KUKA KRL program: Enlargedx2Test.src

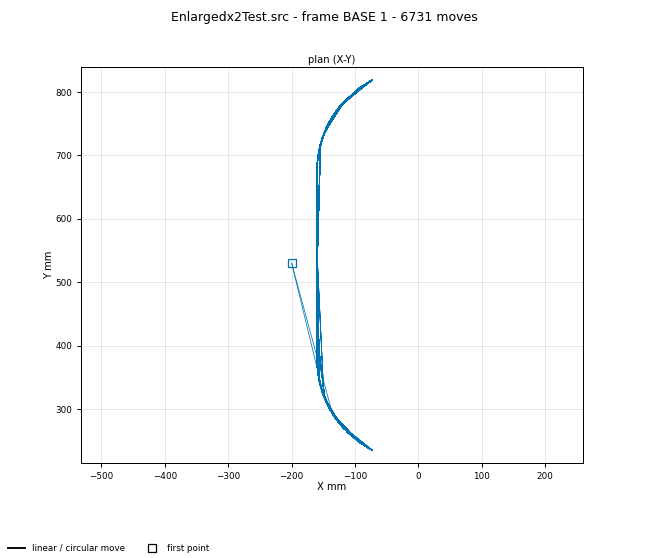
[picture p0: tool path of Enlargedx2Test.src in frame BASE 1, 6731 of 6732 moves have a stored position in this frame; points joined in program order, loops and branches not executed]
&ACCESS RVEO
&REL 11
&PARAM TEMPLATE = C:\KRC\Roboter\Template\vorgabe
&PARAM EDITMASK = *
DEF variable_helical2( )
;FOLD INI
  ;FOLD BASISTECH INI
    GLOBAL INTERRUPT DECL 3 WHEN $STOPMESS==TRUE DO IR_STOPM ( )
    INTERRUPT ON 3
    BAS (#INITMOV,0 )
  ;ENDFOLD (BASISTECH INI)
 ;FOLD USER INI


    ;Make your modifications here
  ;ENDFOLD (USER INI)
;ENDFOLD (INI)
ACTION(#AXIS_RESET,34,1000,#NOERROR,ERROR_CODE)
;FOLD PTP HOME  Vel= 100 % DEFAULT;%{PE}%MKUKATPBASIS,%CMOVE,%VPTP,%P 1:PTP, 2:HOME, 3:, 5:100, 7:DEFAULT
$BWDSTART = FALSE
PDAT_ACT=PDEFAULT
FDAT_ACT=FHOME
BAS (#PTP_PARAMS,100 )
$H_POS=XHOME
PTP  XHOME
;ENDFOLD
BAS(#TOOL,1)
BAS(#BASE,1)
$VEL_AXIS[1]=100
$VEL_AXIS[2]=100
$VEL_AXIS[3]=100
$VEL_AXIS[4]=100
$VEL_AXIS[5]=100
$VEL_AXIS[6]=100
$VEL_EXTAX[1]=100
$VEL_EXTAX[2]=100

$ACC_AXIS[1]=100
$ACC_AXIS[2]=100
$ACC_AXIS[3]=100
$ACC_AXIS[4]=100
$ACC_AXIS[5]=100
$ACC_AXIS[6]=100
$ACC_EXTAX[1]=100
$ACC_EXTAX[2]=100

;;;;;;;;; postprocessing parameters (date 2024-01-29T17:09:42.519984)
; qxconst: -159.99
; qxconstarcys: -152.5,146.5
; qE3offset: 0.00
; qyoffset: 530.00
; qswitchsplit: 3
; qthinningtol: 0.2010
;;;;;;;;;

SLIN {X  -200.000, Y  +530.000, Z    +0.000, A    +0.000, E1    +0.000, E3    +0.000, E4    +0.000}

SLIN {X  -135.697, Y  +292.747, Z    +0.000, E1   +74.259, E3  -294.688}
HALT
SPLINE
SPL {X  -132.590, Y  +287.964, Z    +0.000, E1   +73.910, E3  -289.659}
SPL {X  -129.541, Y  +283.606, Z    +0.000, E1   +73.551, E3  -285.019}
SPL {X  -126.457, Y  +279.493, Z    +0.000, E1   +73.175, E3  -280.620}
SPL {X  -122.770, Y  +274.912, Z    +0.000, E1   +72.712, E3  -275.765}
SPL {X  -119.156, Y  +270.736, Z    +0.000, E1   +72.213, E3  -271.415}
SPL {X  -117.531, Y  +268.949, Z    +0.000, E1   +71.964, E3  -269.600}
SPL {X   -74.907, Y  +236.129, Z    +0.000, E1   +61.720, E3  -192.564}
SPL {X   -72.759, Y  +235.012, Z    +0.000, E1   +56.036, E3   -20.886}
ENDSPLINE

SPLINE
SPL {X  -110.316, Y  +261.624, Z    +0.000, E1   +58.739, E3   +51.186}
SPL {X  -136.558, Y  +294.141, Z    +0.000, E1   +54.887, E3   +72.984}
SPL {X  -153.807, Y  +333.452, Z    +0.000, E1   +40.945, E3   +83.380}
SPL {X  -158.168, Y  +353.421, Z    +0.000, E1   +27.296, E3   +85.774}
SPL {X  -159.556, Y  +365.719, Z    +0.000, E1   +15.845, E3   +86.575}
SPL {X  -159.982, Y  +375.924, Z    +0.000, E1    +4.476, E3   +86.877}
SPL {X  -159.990, Y  +379.800, Z    +0.000, E1    -0.377, E3   +86.905}
SPL {X  -159.990, Y  +383.422, Z    +0.000, E1   -10.730, E3   +86.948}
SPL {X  -159.990, Y  +387.978, Z    +0.000, E1   -23.882, E3   +87.101}
SPL {X  -159.990, Y  +394.494, Z    +0.000, E1   -40.961, E3   +87.482}
SPL {X  -159.990, Y  +400.492, Z    +0.000, E1   -51.837, E3   +88.006}
SPL {X  -159.990, Y  +409.662, Z    +0.000, E1   -61.705, E3   +89.117}
SPL {X  -159.990, Y  +434.697, Z    +0.000, E1   -71.504, E3   +94.137}
SPL {X  -159.990, Y  +521.523, Z    +0.000, E1   -76.035, E3  +120.417}
SPL {X  -154.459, Y  +718.205, Z    +0.000, E1   -76.329, E3  +202.213}
SPL {X  -151.356, Y  +728.349, Z    +0.000, E1   -76.056, E3  +210.428}
SPL {X  -147.124, Y  +739.360, Z    +0.000, E1   -75.690, E3  +220.024}
SPL {X  -142.861, Y  +748.524, Z    +0.000, E1   -75.261, E3  +228.709}
SPL {X  -138.117, Y  +757.250, Z    +0.000, E1   -74.803, E3  +237.313}
SPL {X  -133.491, Y  +764.686, Z    +0.000, E1   -74.276, E3  +245.054}
SPL {X  -130.530, Y  +769.013, Z    +0.000, E1   -73.929, E3  +249.636}
SPL {X  -127.734, Y  +772.837, Z    +0.000, E1   -73.601, E3  +253.688}
SPL {X  -124.765, Y  +776.652, Z    +0.000, E1   -73.233, E3  +257.722}
SPL {X  -121.376, Y  +780.734, Z    +0.000, E1   -72.804, E3  +261.984}
SPL {X  -118.281, Y  +784.233, Z    +0.000, E1   -72.371, E3  +265.552}
SPL {X   -72.391, Y  +819.176, Z    +0.000, E1   -59.867, E3  +361.438}
ENDSPLINE

SPLINE
SPL {X   -92.809, Y  +806.820, Z    +0.000, E1   -56.994, E3  +554.233}
SPL {X  -120.521, Y  +781.721, Z    +0.000, E1   -56.766, E3  +590.332}
SPL {X  -143.482, Y  +747.279, Z    +0.000, E1   -50.227, E3  +608.345}
SPL {X  -154.118, Y  +719.449, Z    +0.000, E1   -38.836, E3  +614.924}
SPL {X  -158.958, Y  +694.646, Z    +0.000, E1   -21.132, E3  +617.775}
SPL {X  -159.960, Y  +679.609, Z    +0.000, E1    -6.021, E3  +618.475}
SPL {X  -159.990, Y  +674.508, Z    +0.000, E1    -0.018, E3  +618.534}
SPL {X  -159.990, Y  +672.787, Z    +0.000, E1    +4.022, E3  +618.546}
SPL {X  -159.990, Y  +669.267, Z    +0.000, E1   +13.665, E3  +618.616}
SPL {X  -159.990, Y  +665.069, Z    +0.000, E1   +25.376, E3  +618.788}
SPL {X  -159.990, Y  +657.821, Z    +0.000, E1   +42.408, E3  +619.290}
SPL {X  -159.990, Y  +645.368, Z    +0.000, E1   +59.257, E3  +620.747}
SPL {X  -159.990, Y  +624.023, Z    +0.000, E1   +69.513, E3  +624.872}
SPL {X  -159.990, Y  +543.075, Z    +0.000, E1   +75.590, E3  +648.520}
SPL {X  -156.121, Y  +342.530, Z    +0.000, E1   +75.868, E3  +735.166}
SPL {X  -153.865, Y  +333.657, Z    +0.000, E1   +75.438, E3  +744.770}
ENDSPLINE

SPLINE
SPL {X  -159.103, Y  +360.678, Z    +0.000, E1   +72.233, E3  +762.874}
ENDSPLINE

SPLINE
SPL {X  -154.371, Y  +335.471, Z    +0.000, E1   +73.016, E3  +771.445}
SPL {X  -148.318, Y  +317.512, Z    +0.000, E1   +73.488, E3  +777.766}
SPL {X  -141.230, Y  +302.327, Z    +0.000, E1   +73.933, E3  +782.319}
SPL {X  -135.697, Y  +292.747, Z    +0.000, E1   +74.259, E3  +784.678}
SPL {X  -132.590, Y  +287.964, Z    +0.000, E1   +73.910, E3  +789.706}
SPL {X  -129.541, Y  +283.606, Z    +0.000, E1   +73.551, E3  +794.346}
SPL {X  -126.457, Y  +279.493, Z    +0.000, E1   +73.175, E3  +798.745}
SPL {X  -122.770, Y  +274.912, Z    +0.000, E1   +72.712, E3  +803.600}
SPL {X  -119.156, Y  +270.736, Z    +0.000, E1   +72.213, E3  +807.950}
SPL {X  -117.531, Y  +268.949, Z    +0.000, E1   +71.964, E3  +809.765}
SPL {X   -74.907, Y  +236.129, Z    +0.000, E1   +61.720, E3  +886.801}
SPL {X   -72.759, Y  +235.012, Z    +0.000, E1   +56.036, E3 +1058.479}
ENDSPLINE

SPLINE
SPL {X  -110.316, Y  +261.624, Z    +0.000, E1   +58.739, E3 +1130.551}
SPL {X  -136.558, Y  +294.141, Z    +0.000, E1   +54.887, E3 +1152.349}
SPL {X  -153.807, Y  +333.452, Z    +0.000, E1   +40.945, E3 +1162.745}
SPL {X  -158.168, Y  +353.421, Z    +0.000, E1   +27.296, E3 +1165.139}
SPL {X  -159.556, Y  +365.719, Z    +0.000, E1   +15.845, E3 +1165.940}
SPL {X  -159.982, Y  +375.924, Z    +0.000, E1    +4.476, E3 +1166.242}
SPL {X  -159.990, Y  +379.800, Z    +0.000, E1    -0.377, E3 +1166.270}
SPL {X  -159.990, Y  +383.422, Z    +0.000, E1   -10.730, E3 +1166.313}
SPL {X  -159.990, Y  +387.978, Z    +0.000, E1   -23.882, E3 +1166.466}
SPL {X  -159.990, Y  +394.494, Z    +0.000, E1   -40.961, E3 +1166.847}
SPL {X  -159.990, Y  +400.492, Z    +0.000, E1   -51.837, E3 +1167.371}
SPL {X  -159.990, Y  +409.662, Z    +0.000, E1   -61.705, E3 +1168.482}
SPL {X  -159.990, Y  +434.697, Z    +0.000, E1   -71.504, E3 +1173.502}
SPL {X  -159.990, Y  +521.523, Z    +0.000, E1   -76.035, E3 +1199.782}
SPL {X  -154.459, Y  +718.205, Z    +0.000, E1   -76.329, E3 +1281.578}
SPL {X  -151.356, Y  +728.349, Z    +0.000, E1   -76.056, E3 +1289.793}
SPL {X  -147.124, Y  +739.360, Z    +0.000, E1   -75.690, E3 +1299.390}
SPL {X  -142.861, Y  +748.524, Z    +0.000, E1   -75.261, E3 +1308.074}
SPL {X  -138.117, Y  +757.250, Z    +0.000, E1   -74.803, E3 +1316.678}
SPL {X  -133.491, Y  +764.686, Z    +0.000, E1   -74.276, E3 +1324.419}
SPL {X  -130.530, Y  +769.013, Z    +0.000, E1   -73.929, E3 +1329.001}
SPL {X  -127.734, Y  +772.837, Z    +0.000, E1   -73.601, E3 +1333.053}
SPL {X  -124.765, Y  +776.652, Z    +0.000, E1   -73.233, E3 +1337.087}
SPL {X  -121.376, Y  +780.734, Z    +0.000, E1   -72.804, E3 +1341.349}
SPL {X  -118.281, Y  +784.233, Z    +0.000, E1   -72.371, E3 +1344.917}
SPL {X   -72.391, Y  +819.176, Z    +0.000, E1   -59.867, E3 +1440.803}
ENDSPLINE

SPLINE
SPL {X  -116.241, Y  +786.431, Z    +0.000, E1   -57.120, E3 +1665.245}
SPL {X  -148.710, Y  +735.509, Z    +0.000, E1   -46.282, E3 +1690.978}
SPL {X  -157.559, Y  +704.285, Z    +0.000, E1   -29.037, E3 +1696.307}
SPL {X  -159.430, Y  +689.871, Z    +0.000, E1   -16.582, E3 +1697.457}
SPL {X  -159.960, Y  +679.609, Z    +0.000, E1    -6.021, E3 +1697.841}
SPL {X  -159.990, Y  +674.508, Z    +0.000, E1    -0.018, E3 +1697.899}
SPL {X  -159.990, Y  +672.787, Z    +0.000, E1    +4.022, E3 +1697.911}
SPL {X  -159.990, Y  +669.267, Z    +0.000, E1   +13.665, E3 +1697.981}
SPL {X  -159.990, Y  +663.438, Z    +0.000, E1   +29.379, E3 +1698.252}
SPL {X  -159.990, Y  +655.264, Z    +0.000, E1   +47.291, E3 +1698.869}
SPL {X  -159.990, Y  +645.368, Z    +0.000, E1   +59.257, E3 +1700.112}
SPL {X  -159.990, Y  +624.023, Z    +0.000, E1   +69.513, E3 +1704.237}
SPL {X  -159.990, Y  +543.075, Z    +0.000, E1   +75.590, E3 +1727.885}
SPL {X  -156.121, Y  +342.530, Z    +0.000, E1   +75.868, E3 +1814.531}
SPL {X  -153.498, Y  +332.386, Z    +0.000, E1   +75.628, E3 +1822.536}
ENDSPLINE

SPLINE
SPL {X  -155.252, Y  +338.851, Z    +0.000, E1   +74.632, E3 +1829.914}
SPL {X  -159.103, Y  +360.678, Z    +0.000, E1   +72.233, E3 +1842.239}
ENDSPLINE

SPLINE
SPL {X  -154.371, Y  +335.471, Z    +0.000, E1   +73.016, E3 +1850.810}
SPL {X  -149.938, Y  +321.685, Z    +0.000, E1   +73.398, E3 +1855.504}
SPL {X  -145.016, Y  +309.920, Z    +0.000, E1   +73.647, E3 +1860.025}
SPL {X  -139.138, Y  +298.522, Z    +0.000, E1   +74.138, E3 +1862.041}
SPL {X  -135.697, Y  +292.747, Z    +0.000, E1   +74.259, E3 +1864.043}
SPL {X  -132.590, Y  +287.964, Z    +0.000, E1   +73.910, E3 +1869.071}
SPL {X  -129.541, Y  +283.606, Z    +0.000, E1   +73.551, E3 +1873.711}
SPL {X  -126.457, Y  +279.493, Z    +0.000, E1   +73.175, E3 +1878.110}
SPL {X  -122.770, Y  +274.912, Z    +0.000, E1   +72.712, E3 +1882.966}
SPL {X  -119.156, Y  +270.736, Z    +0.000, E1   +72.213, E3 +1887.315}
SPL {X  -117.531, Y  +268.949, Z    +0.000, E1   +71.964, E3 +1889.130}
SPL {X   -74.907, Y  +236.129, Z    +0.000, E1   +61.720, E3 +1966.166}
ENDSPLINE

SPLINE
SPL {X   -94.059, Y  +248.080, Z    +0.000, E1   +58.275, E3 +2187.859}
SPL {X  -130.769, Y  +285.325, Z    +0.000, E1   +56.495, E3 +2227.736}
SPL {X  -149.689, Y  +321.019, Z    +0.000, E1   +46.817, E3 +2239.820}
SPL {X  -157.484, Y  +349.293, Z    +0.000, E1   +30.654, E3 +2244.113}
SPL {X  -159.556, Y  +365.719, Z    +0.000, E1   +15.845, E3 +2245.305}
SPL {X  -159.982, Y  +375.924, Z    +0.000, E1    +4.476, E3 +2245.607}
SPL {X  -159.990, Y  +379.531, Z    +0.000, E1    -0.039, E3 +2245.634}
SPL {X  -159.990, Y  +382.420, Z    +0.000, E1    -7.600, E3 +2245.662}
SPL {X  -159.990, Y  +386.504, Z    +0.000, E1   -19.860, E3 +2245.768}
SPL {X  -159.990, Y  +392.530, Z    +0.000, E1   -36.133, E3 +2246.083}
SPL {X  -159.990, Y  +400.492, Z    +0.000, E1   -51.837, E3 +2246.736}
SPL {X  -159.990, Y  +409.662, Z    +0.000, E1   -61.705, E3 +2247.847}
SPL {X  -159.990, Y  +434.697, Z    +0.000, E1   -71.504, E3 +2252.867}
SPL {X  -159.990, Y  +521.523, Z    +0.000, E1   -76.035, E3 +2279.148}
SPL {X  -154.459, Y  +718.205, Z    +0.000, E1   -76.329, E3 +2360.943}
SPL {X  -151.356, Y  +728.349, Z    +0.000, E1   -76.056, E3 +2369.158}
SPL {X  -148.399, Y  +736.287, Z    +0.000, E1   -75.788, E3 +2376.037}
SPL {X  -144.005, Y  +746.209, Z    +0.000, E1   -75.396, E3 +2385.153}
SPL {X  -138.117, Y  +757.250, Z    +0.000, E1   -74.803, E3 +2396.043}
SPL {X  -133.491, Y  +764.686, Z    +0.000, E1   -74.276, E3 +2403.784}
SPL {X  -128.839, Y  +771.354, Z    +0.000, E1   -73.759, E3 +2410.803}
SPL {X  -123.568, Y  +778.125, Z    +0.000, E1   -73.105, E3 +2417.974}
SPL {X  -118.985, Y  +783.455, Z    +0.000, E1   -72.490, E3 +2423.482}
SPL {X   -72.391, Y  +819.176, Z    +0.000, E1   -59.867, E3 +2520.168}
ENDSPLINE

SPLINE
SPL {X   -92.809, Y  +806.820, Z    +0.000, E1   -56.994, E3 +2712.963}
SPL {X  -120.521, Y  +781.721, Z    +0.000, E1   -56.766, E3 +2749.062}
SPL {X  -143.482, Y  +747.279, Z    +0.000, E1   -50.227, E3 +2767.075}
SPL {X  -154.118, Y  +719.449, Z    +0.000, E1   -38.836, E3 +2773.654}
SPL {X  -158.958, Y  +694.646, Z    +0.000, E1   -21.132, E3 +2776.506}
SPL {X  -159.960, Y  +679.609, Z    +0.000, E1    -6.021, E3 +2777.206}
SPL {X  -159.990, Y  +674.508, Z    +0.000, E1    -0.018, E3 +2777.264}
SPL {X  -159.990, Y  +672.787, Z    +0.000, E1    +4.022, E3 +2777.276}
SPL {X  -159.990, Y  +669.267, Z    +0.000, E1   +13.665, E3 +2777.346}
SPL {X  -159.990, Y  +663.438, Z    +0.000, E1   +29.379, E3 +2777.617}
SPL {X  -159.990, Y  +655.264, Z    +0.000, E1   +47.291, E3 +2778.234}
SPL {X  -159.990, Y  +645.368, Z    +0.000, E1   +59.257, E3 +2779.477}
SPL {X  -159.990, Y  +624.023, Z    +0.000, E1   +69.513, E3 +2783.602}
SPL {X  -159.990, Y  +543.075, Z    +0.000, E1   +75.590, E3 +2807.250}
SPL {X  -156.121, Y  +342.530, Z    +0.000, E1   +75.868, E3 +2893.896}
SPL {X  -153.498, Y  +332.386, Z    +0.000, E1   +75.628, E3 +2901.901}
ENDSPLINE

SPLINE
SPL {X  -155.252, Y  +338.851, Z    +0.000, E1   +74.632, E3 +2909.279}
SPL {X  -159.103, Y  +360.678, Z    +0.000, E1   +72.233, E3 +2921.604}
ENDSPLINE

SPLINE
SPL {X  -154.371, Y  +335.471, Z    +0.000, E1   +73.016, E3 +2930.175}
SPL {X  -149.938, Y  +321.685, Z    +0.000, E1   +73.398, E3 +2934.869}
SPL {X  -145.016, Y  +309.920, Z    +0.000, E1   +73.647, E3 +2939.390}
SPL {X  -139.138, Y  +298.522, Z    +0.000, E1   +74.138, E3 +2941.406}
SPL {X  -135.697, Y  +292.747, Z    +0.000, E1   +74.259, E3 +2943.408}
SPL {X  -132.590, Y  +287.964, Z    +0.000, E1   +73.910, E3 +2948.436}
SPL {X  -129.541, Y  +283.606, Z    +0.000, E1   +73.551, E3 +2953.076}
SPL {X  -126.457, Y  +279.493, Z    +0.000, E1   +73.175, E3 +2957.475}
SPL {X  -122.770, Y  +274.912, Z    +0.000, E1   +72.712, E3 +2962.331}
SPL {X  -118.941, Y  +270.496, Z    +0.000, E1   +72.188, E3 +2966.918}
SPL {X   -74.907, Y  +236.129, Z    +0.000, E1   +61.720, E3 +3045.531}
ENDSPLINE

SPLINE
SPL {X   -94.059, Y  +248.080, Z    +0.000, E1   +58.275, E3 +3267.224}
SPL {X  -136.558, Y  +294.141, Z    +0.000, E1   +54.887, E3 +3311.079}
SPL {X  -151.843, Y  +327.098, Z    +0.000, E1   +44.118, E3 +3320.438}
SPL {X  -157.484, Y  +349.293, Z    +0.000, E1   +30.654, E3 +3323.478}
SPL {X  -159.556, Y  +365.719, Z    +0.000, E1   +15.845, E3 +3324.670}
SPL {X  -159.982, Y  +375.924, Z    +0.000, E1    +4.476, E3 +3324.972}
SPL {X  -159.990, Y  +379.531, Z    +0.000, E1    -0.039, E3 +3324.999}
SPL {X  -159.990, Y  +382.420, Z    +0.000, E1    -7.600, E3 +3325.027}
SPL {X  -159.990, Y  +386.504, Z    +0.000, E1   -19.860, E3 +3325.133}
SPL {X  -159.990, Y  +392.530, Z    +0.000, E1   -36.133, E3 +3325.448}
SPL {X  -159.990, Y  +400.492, Z    +0.000, E1   -51.837, E3 +3326.101}
SPL {X  -159.990, Y  +409.662, Z    +0.000, E1   -61.705, E3 +3327.212}
SPL {X  -159.990, Y  +434.697, Z    +0.000, E1   -71.504, E3 +3332.232}
SPL {X  -159.990, Y  +521.523, Z    +0.000, E1   -76.035, E3 +3358.513}
SPL {X  -154.459, Y  +718.205, Z    +0.000, E1   -76.329, E3 +3440.308}
SPL {X  -151.356, Y  +728.349, Z    +0.000, E1   -76.056, E3 +3448.523}
SPL {X  -148.399, Y  +736.287, Z    +0.000, E1   -75.788, E3 +3455.402}
SPL {X  -144.005, Y  +746.209, Z    +0.000, E1   -75.396, E3 +3464.518}
SPL {X  -138.117, Y  +757.250, Z    +0.000, E1   -74.803, E3 +3475.408}
SPL {X  -133.491, Y  +764.686, Z    +0.000, E1   -74.276, E3 +3483.149}
SPL {X  -128.839, Y  +771.354, Z    +0.000, E1   -73.759, E3 +3490.168}
SPL {X  -123.568, Y  +778.125, Z    +0.000, E1   -73.105, E3 +3497.339}
SPL {X  -118.985, Y  +783.455, Z    +0.000, E1   -72.490, E3 +3502.847}
SPL {X   -72.391, Y  +819.176, Z    +0.000, E1   -59.867, E3 +3599.533}
ENDSPLINE

SPLINE
SPL {X   -92.809, Y  +806.820, Z    +0.000, E1   -56.994, E3 +3792.328}
SPL {X  -120.521, Y  +781.721, Z    +0.000, E1   -56.766, E3 +3828.427}
SPL {X  -148.710, Y  +735.509, Z    +0.000, E1   -46.282, E3 +3849.708}
SPL {X  -157.559, Y  +704.285, Z    +0.000, E1   -29.037, E3 +3855.037}
SPL {X  -159.430, Y  +689.871, Z    +0.000, E1   -16.582, E3 +3856.188}
SPL {X  -159.960, Y  +679.609, Z    +0.000, E1    -6.021, E3 +3856.571}
SPL {X  -159.990, Y  +674.508, Z    +0.000, E1    -0.018, E3 +3856.629}
SPL {X  -159.990, Y  +672.787, Z    +0.000, E1    +4.022, E3 +3856.641}
SPL {X  -159.990, Y  +669.267, Z    +0.000, E1   +13.665, E3 +3856.711}
SPL {X  -159.990, Y  +663.438, Z    +0.000, E1   +29.379, E3 +3856.982}
SPL {X  -159.990, Y  +655.264, Z    +0.000, E1   +47.291, E3 +3857.599}
SPL {X  -159.990, Y  +645.368, Z    +0.000, E1   +59.257, E3 +3858.842}
SPL {X  -159.990, Y  +624.023, Z    +0.000, E1   +69.513, E3 +3862.967}
SPL {X  -159.990, Y  +543.075, Z    +0.000, E1   +75.590, E3 +3886.615}
SPL {X  -156.121, Y  +342.530, Z    +0.000, E1   +75.868, E3 +3973.261}
SPL {X  -153.865, Y  +333.657, Z    +0.000, E1   +75.438, E3 +3982.865}
ENDSPLINE

SPLINE
SPL {X  -159.644, Y  +366.989, Z    +0.000, E1   +72.058, E3 +3998.392}
ENDSPLINE

SPLINE
SPL {X  -156.933, Y  +346.374, Z    +0.000, E1   +72.645, E3 +4006.281}
SPL {X  -151.144, Y  +325.039, Z    +0.000, E1   +73.323, E3 +4012.961}
SPL {X  -145.016, Y  +309.920, Z    +0.000, E1   +73.647, E3 +4018.755}
SPL {X  -136.944, Y  +294.777, Z    +0.000, E1   +74.219, E3 +4022.057}
SPL {X  -132.590, Y  +287.964, Z    +0.000, E1   +73.910, E3 +4027.801}
SPL {X  -129.541, Y  +283.606, Z    +0.000, E1   +73.551, E3 +4032.441}
SPL {X  -125.403, Y  +278.147, Z    +0.000, E1   +73.063, E3 +4038.249}
SPL {X  -121.908, Y  +273.889, Z    +0.000, E1   +72.578, E3 +4042.795}
SPL {X  -118.941, Y  +270.496, Z    +0.000, E1   +72.188, E3 +4046.283}
SPL {X   -74.907, Y  +236.129, Z    +0.000, E1   +61.720, E3 +4124.897}
ENDSPLINE

SPLINE
SPL {X   -94.059, Y  +248.080, Z    +0.000, E1   +58.275, E3 +4346.589}
SPL {X  -136.558, Y  +294.141, Z    +0.000, E1   +54.887, E3 +4390.444}
SPL {X  -151.843, Y  +327.098, Z    +0.000, E1   +44.118, E3 +4399.804}
SPL {X  -157.484, Y  +349.293, Z    +0.000, E1   +30.654, E3 +4402.843}
SPL {X  -159.556, Y  +365.719, Z    +0.000, E1   +15.845, E3 +4404.035}
SPL {X  -159.982, Y  +375.924, Z    +0.000, E1    +4.476, E3 +4404.337}
SPL {X  -159.990, Y  +379.531, Z    +0.000, E1    -0.039, E3 +4404.364}
SPL {X  -159.990, Y  +382.420, Z    +0.000, E1    -7.600, E3 +4404.393}
SPL {X  -159.990, Y  +386.504, Z    +0.000, E1   -19.860, E3 +4404.498}
SPL {X  -159.990, Y  +392.530, Z    +0.000, E1   -36.133, E3 +4404.813}
SPL {X  -159.990, Y  +400.492, Z    +0.000, E1   -51.837, E3 +4405.466}
SPL {X  -159.990, Y  +409.662, Z    +0.000, E1   -61.705, E3 +4406.577}
SPL {X  -159.990, Y  +434.697, Z    +0.000, E1   -71.504, E3 +4411.597}
SPL {X  -159.990, Y  +521.523, Z    +0.000, E1   -76.035, E3 +4437.878}
SPL {X  -154.459, Y  +718.205, Z    +0.000, E1   -76.329, E3 +4519.673}
SPL {X  -151.356, Y  +728.349, Z    +0.000, E1   -76.056, E3 +4527.889}
SPL {X  -148.399, Y  +736.287, Z    +0.000, E1   -75.788, E3 +4534.767}
SPL {X  -144.005, Y  +746.209, Z    +0.000, E1   -75.396, E3 +4543.883}
SPL {X  -138.117, Y  +757.250, Z    +0.000, E1   -74.803, E3 +4554.773}
SPL {X  -133.491, Y  +764.686, Z    +0.000, E1   -74.276, E3 +4562.514}
SPL {X  -128.839, Y  +771.354, Z    +0.000, E1   -73.759, E3 +4569.533}
SPL {X  -123.568, Y  +778.125, Z    +0.000, E1   -73.105, E3 +4576.705}
SPL {X  -118.985, Y  +783.455, Z    +0.000, E1   -72.490, E3 +4582.212}
SPL {X   -72.391, Y  +819.176, Z    +0.000, E1   -59.867, E3 +4678.898}
ENDSPLINE

SPLINE
SPL {X   -92.809, Y  +806.820, Z    +0.000, E1   -56.994, E3 +4871.693}
SPL {X  -120.521, Y  +781.721, Z    +0.000, E1   -56.766, E3 +4907.792}
SPL {X  -143.482, Y  +747.279, Z    +0.000, E1   -50.227, E3 +4925.805}
SPL {X  -154.118, Y  +719.449, Z    +0.000, E1   -38.836, E3 +4932.384}
SPL {X  -158.958, Y  +694.646, Z    +0.000, E1   -21.132, E3 +4935.236}
SPL {X  -159.960, Y  +679.609, Z    +0.000, E1    -6.021, E3 +4935.936}
SPL {X  -159.990, Y  +674.508, Z    +0.000, E1    -0.018, E3 +4935.994}
SPL {X  -159.990, Y  +672.787, Z    +0.000, E1    +4.022, E3 +4936.006}
SPL {X  -159.990, Y  +669.267, Z    +0.000, E1   +13.665, E3 +4936.076}
SPL {X  -159.990, Y  +663.438, Z    +0.000, E1   +29.379, E3 +4936.347}
SPL {X  -159.990, Y  +655.264, Z    +0.000, E1   +47.291, E3 +4936.964}
SPL {X  -159.990, Y  +645.368, Z    +0.000, E1   +59.257, E3 +4938.207}
SPL {X  -159.990, Y  +624.023, Z    +0.000, E1   +69.513, E3 +4942.332}
SPL {X  -159.990, Y  +543.075, Z    +0.000, E1   +75.590, E3 +4965.980}
SPL {X  -156.121, Y  +342.530, Z    +0.000, E1   +75.868, E3 +5052.626}
SPL {X  -153.498, Y  +332.386, Z    +0.000, E1   +75.628, E3 +5060.631}
ENDSPLINE

SPLINE
SPL {X  -155.252, Y  +338.851, Z    +0.000, E1   +74.632, E3 +5068.009}
SPL {X  -159.103, Y  +360.678, Z    +0.000, E1   +72.233, E3 +5080.334}
ENDSPLINE

SPLINE
SPL {X  -154.371, Y  +335.471, Z    +0.000, E1   +73.016, E3 +5088.905}
SPL {X  -149.938, Y  +321.685, Z    +0.000, E1   +73.398, E3 +5093.599}
SPL {X  -145.016, Y  +309.920, Z    +0.000, E1   +73.647, E3 +5098.120}
SPL {X  -139.138, Y  +298.522, Z    +0.000, E1   +74.138, E3 +5100.136}
SPL {X  -135.697, Y  +292.747, Z    +0.000, E1   +74.259, E3 +5102.138}
SPL {X  -132.590, Y  +287.964, Z    +0.000, E1   +73.910, E3 +5107.166}
SPL {X  -129.541, Y  +283.606, Z    +0.000, E1   +73.551, E3 +5111.807}
SPL {X  -126.457, Y  +279.493, Z    +0.000, E1   +73.175, E3 +5116.206}
SPL {X  -122.770, Y  +274.912, Z    +0.000, E1   +72.712, E3 +5121.061}
SPL {X  -118.941, Y  +270.496, Z    +0.000, E1   +72.188, E3 +5125.648}
SPL {X   -74.907, Y  +236.129, Z    +0.000, E1   +61.720, E3 +5204.262}
ENDSPLINE

SPLINE
SPL {X   -94.059, Y  +248.080, Z    +0.000, E1   +58.275, E3 +5425.955}
SPL {X  -136.558, Y  +294.141, Z    +0.000, E1   +54.887, E3 +5469.809}
SPL {X  -151.843, Y  +327.098, Z    +0.000, E1   +44.118, E3 +5479.169}
SPL {X  -157.484, Y  +349.293, Z    +0.000, E1   +30.654, E3 +5482.208}
SPL {X  -159.556, Y  +365.719, Z    +0.000, E1   +15.845, E3 +5483.401}
SPL {X  -159.982, Y  +375.924, Z    +0.000, E1    +4.476, E3 +5483.702}
SPL {X  -159.990, Y  +379.531, Z    +0.000, E1    -0.039, E3 +5483.729}
SPL {X  -159.990, Y  +382.420, Z    +0.000, E1    -7.600, E3 +5483.758}
SPL {X  -159.990, Y  +386.504, Z    +0.000, E1   -19.860, E3 +5483.863}
SPL {X  -159.990, Y  +392.530, Z    +0.000, E1   -36.133, E3 +5484.178}
SPL {X  -159.990, Y  +400.492, Z    +0.000, E1   -51.837, E3 +5484.831}
SPL {X  -159.990, Y  +409.662, Z    +0.000, E1   -61.705, E3 +5485.942}
SPL {X  -159.990, Y  +434.697, Z    +0.000, E1   -71.504, E3 +5490.962}
SPL {X  -159.990, Y  +521.523, Z    +0.000, E1   -76.035, E3 +5517.243}
SPL {X  -154.459, Y  +718.205, Z    +0.000, E1   -76.329, E3 +5599.038}
SPL {X  -151.356, Y  +728.349, Z    +0.000, E1   -76.056, E3 +5607.254}
SPL {X  -148.399, Y  +736.287, Z    +0.000, E1   -75.788, E3 +5614.132}
SPL {X  -144.005, Y  +746.209, Z    +0.000, E1   -75.396, E3 +5623.248}
SPL {X  -138.117, Y  +757.250, Z    +0.000, E1   -74.803, E3 +5634.138}
SPL {X  -133.491, Y  +764.686, Z    +0.000, E1   -74.276, E3 +5641.879}
SPL {X  -128.839, Y  +771.354, Z    +0.000, E1   -73.759, E3 +5648.898}
SPL {X  -123.568, Y  +778.125, Z    +0.000, E1   -73.105, E3 +5656.070}
SPL {X  -118.985, Y  +783.455, Z    +0.000, E1   -72.490, E3 +5661.577}
SPL {X   -72.391, Y  +819.176, Z    +0.000, E1   -59.867, E3 +5758.263}
ENDSPLINE

SPLINE
SPL {X   -92.809, Y  +806.820, Z    +0.000, E1   -56.994, E3 +5951.058}
SPL {X  -120.521, Y  +781.721, Z    +0.000, E1   -56.766, E3 +5987.157}
SPL {X  -148.710, Y  +735.509, Z    +0.000, E1   -46.282, E3 +6008.438}
SPL {X  -157.559, Y  +704.285, Z    +0.000, E1   -29.037, E3 +6013.768}
SPL {X  -159.430, Y  +689.871, Z    +0.000, E1   -16.582, E3 +6014.918}
SPL {X  -159.960, Y  +679.609, Z    +0.000, E1    -6.021, E3 +6015.301}
SPL {X  -159.990, Y  +674.508, Z    +0.000, E1    -0.018, E3 +6015.360}
SPL {X  -159.990, Y  +672.787, Z    +0.000, E1    +4.022, E3 +6015.371}
SPL {X  -159.990, Y  +669.267, Z    +0.000, E1   +13.665, E3 +6015.442}
SPL {X  -159.990, Y  +663.438, Z    +0.000, E1   +29.379, E3 +6015.712}
SPL {X  -159.990, Y  +655.264, Z    +0.000, E1   +47.291, E3 +6016.329}
SPL {X  -159.990, Y  +645.368, Z    +0.000, E1   +59.257, E3 +6017.572}
SPL {X  -159.990, Y  +624.023, Z    +0.000, E1   +69.513, E3 +6021.697}
SPL {X  -159.990, Y  +543.075, Z    +0.000, E1   +75.590, E3 +6045.345}
SPL {X  -156.121, Y  +342.530, Z    +0.000, E1   +75.868, E3 +6131.991}
SPL {X  -153.865, Y  +333.657, Z    +0.000, E1   +75.438, E3 +6141.595}
ENDSPLINE

SPLINE
SPL {X  -159.644, Y  +366.989, Z    +0.000, E1   +72.058, E3 +6157.122}
ENDSPLINE

SPLINE
SPL {X  -156.933, Y  +346.374, Z    +0.000, E1   +72.645, E3 +6165.012}
SPL {X  -151.144, Y  +325.039, Z    +0.000, E1   +73.323, E3 +6171.691}
SPL {X  -146.668, Y  +313.584, Z    +0.000, E1   +73.560, E3 +6176.173}
SPL {X  -141.230, Y  +302.327, Z    +0.000, E1   +73.933, E3 +6179.145}
SPL {X  -135.697, Y  +292.747, Z    +0.000, E1   +74.259, E3 +6181.503}
SPL {X  -132.590, Y  +287.964, Z    +0.000, E1   +73.910, E3 +6186.531}
SPL {X  -129.541, Y  +283.606, Z    +0.000, E1   +73.551, E3 +6191.172}
SPL {X  -125.403, Y  +278.147, Z    +0.000, E1   +73.063, E3 +6196.979}
SPL {X  -121.908, Y  +273.889, Z    +0.000, E1   +72.578, E3 +6201.525}
SPL {X  -119.156, Y  +270.736, Z    +0.000, E1   +72.213, E3 +6204.775}
SPL {X  -117.531, Y  +268.949, Z    +0.000, E1   +71.964, E3 +6206.591}
SPL {X   -74.907, Y  +236.129, Z    +0.000, E1   +61.720, E3 +6283.627}
ENDSPLINE

SPLINE
SPL {X   -94.059, Y  +248.080, Z    +0.000, E1   +58.275, E3 +6505.320}
SPL {X  -130.769, Y  +285.325, Z    +0.000, E1   +56.495, E3 +6545.197}
SPL {X  -149.689, Y  +321.019, Z    +0.000, E1   +46.817, E3 +6557.281}
SPL {X  -157.484, Y  +349.293, Z    +0.000, E1   +30.654, E3 +6561.573}
SPL {X  -159.556, Y  +365.719, Z    +0.000, E1   +15.845, E3 +6562.766}
SPL {X  -159.982, Y  +375.924, Z    +0.000, E1    +4.476, E3 +6563.067}
SPL {X  -159.990, Y  +379.531, Z    +0.000, E1    -0.039, E3 +6563.094}
SPL {X  -159.990, Y  +382.420, Z    +0.000, E1    -7.600, E3 +6563.123}
SPL {X  -159.990, Y  +386.504, Z    +0.000, E1   -19.860, E3 +6563.228}
SPL {X  -159.990, Y  +392.530, Z    +0.000, E1   -36.133, E3 +6563.543}
SPL {X  -159.990, Y  +400.492, Z    +0.000, E1   -51.837, E3 +6564.196}
SPL {X  -159.990, Y  +409.662, Z    +0.000, E1   -61.705, E3 +6565.307}
SPL {X  -159.990, Y  +434.697, Z    +0.000, E1   -71.504, E3 +6570.327}
SPL {X  -159.990, Y  +521.523, Z    +0.000, E1   -76.035, E3 +6596.608}
SPL {X  -154.459, Y  +718.205, Z    +0.000, E1   -76.329, E3 +6678.403}
SPL {X  -151.356, Y  +728.349, Z    +0.000, E1   -76.056, E3 +6686.619}
SPL {X  -147.124, Y  +739.360, Z    +0.000, E1   -75.690, E3 +6696.215}
SPL {X  -142.861, Y  +748.524, Z    +0.000, E1   -75.261, E3 +6704.900}
SPL {X  -139.796, Y  +754.307, Z    +0.000, E1   -74.951, E3 +6710.588}
SPL {X  -136.850, Y  +759.378, Z    +0.000, E1   -74.643, E3 +6715.732}
SPL {X  -133.491, Y  +764.686, Z    +0.000, E1   -74.276, E3 +6721.244}
SPL {X  -130.530, Y  +769.013, Z    +0.000, E1   -73.929, E3 +6725.826}
SPL {X  -127.734, Y  +772.837, Z    +0.000, E1   -73.601, E3 +6729.878}
SPL {X  -124.765, Y  +776.652, Z    +0.000, E1   -73.233, E3 +6733.913}
SPL {X  -121.376, Y  +780.734, Z    +0.000, E1   -72.804, E3 +6738.174}
SPL {X  -118.281, Y  +784.233, Z    +0.000, E1   -72.371, E3 +6741.743}
SPL {X   -72.391, Y  +819.176, Z    +0.000, E1   -59.867, E3 +6837.628}
ENDSPLINE

SPLINE
SPL {X  -116.241, Y  +786.431, Z    +0.000, E1   -57.120, E3 +7062.071}
SPL {X  -143.482, Y  +747.279, Z    +0.000, E1   -50.227, E3 +7084.535}
SPL {X  -154.118, Y  +719.449, Z    +0.000, E1   -38.836, E3 +7091.115}
SPL {X  -158.958, Y  +694.646, Z    +0.000, E1   -21.132, E3 +7093.966}
SPL {X  -159.960, Y  +679.609, Z    +0.000, E1    -6.021, E3 +7094.666}
SPL {X  -159.990, Y  +674.508, Z    +0.000, E1    -0.018, E3 +7094.725}
SPL {X  -159.990, Y  +672.787, Z    +0.000, E1    +4.022, E3 +7094.736}
SPL {X  -159.990, Y  +669.267, Z    +0.000, E1   +13.665, E3 +7094.807}
SPL {X  -159.990, Y  +665.069, Z    +0.000, E1   +25.376, E3 +7094.978}
SPL {X  -159.990, Y  +657.821, Z    +0.000, E1   +42.408, E3 +7095.481}
SPL {X  -159.990, Y  +645.368, Z    +0.000, E1   +59.257, E3 +7096.937}
SPL {X  -159.990, Y  +624.023, Z    +0.000, E1   +69.513, E3 +7101.062}
SPL {X  -159.990, Y  +543.075, Z    +0.000, E1   +75.590, E3 +7124.710}
SPL {X  -156.121, Y  +342.530, Z    +0.000, E1   +75.868, E3 +7211.357}
SPL {X  -153.865, Y  +333.657, Z    +0.000, E1   +75.438, E3 +7220.961}
ENDSPLINE

SPLINE
SPL {X  -159.644, Y  +366.989, Z    +0.000, E1   +72.058, E3 +7236.487}
ENDSPLINE

SPLINE
SPL {X  -156.933, Y  +346.374, Z    +0.000, E1   +72.645, E3 +7244.377}
SPL {X  -151.144, Y  +325.039, Z    +0.000, E1   +73.323, E3 +7251.056}
SPL {X  -145.016, Y  +309.920, Z    +0.000, E1   +73.647, E3 +7256.850}
SPL {X  -136.944, Y  +294.777, Z    +0.000, E1   +74.219, E3 +7260.152}
SPL {X  -132.590, Y  +287.964, Z    +0.000, E1   +73.910, E3 +7265.896}
SPL {X  -129.541, Y  +283.606, Z    +0.000, E1   +73.551, E3 +7270.537}
SPL {X  -126.457, Y  +279.493, Z    +0.000, E1   +73.175, E3 +7274.936}
SPL {X  -122.770, Y  +274.912, Z    +0.000, E1   +72.712, E3 +7279.791}
SPL {X  -119.156, Y  +270.736, Z    +0.000, E1   +72.213, E3 +7284.140}
SPL {X  -117.531, Y  +268.949, Z    +0.000, E1   +71.964, E3 +7285.956}
SPL {X   -74.907, Y  +236.129, Z    +0.000, E1   +61.720, E3 +7362.992}
ENDSPLINE

SPLINE
SPL {X   -94.059, Y  +248.080, Z    +0.000, E1   +58.275, E3 +7584.685}
SPL {X  -130.769, Y  +285.325, Z    +0.000, E1   +56.495, E3 +7624.562}
SPL {X  -149.689, Y  +321.019, Z    +0.000, E1   +46.817, E3 +7636.646}
SPL {X  -157.484, Y  +349.293, Z    +0.000, E1   +30.654, E3 +7640.938}
SPL {X  -159.556, Y  +365.719, Z    +0.000, E1   +15.845, E3 +7642.131}
SPL {X  -159.982, Y  +375.924, Z    +0.000, E1    +4.476, E3 +7642.432}
SPL {X  -159.990, Y  +379.531, Z    +0.000, E1    -0.039, E3 +7642.459}
SPL {X  -159.990, Y  +382.420, Z    +0.000, E1    -7.600, E3 +7642.488}
SPL {X  -159.990, Y  +386.504, Z    +0.000, E1   -19.860, E3 +7642.593}
SPL {X  -159.990, Y  +392.530, Z    +0.000, E1   -36.133, E3 +7642.908}
SPL {X  -159.990, Y  +400.492, Z    +0.000, E1   -51.837, E3 +7643.561}
SPL {X  -159.990, Y  +409.662, Z    +0.000, E1   -61.705, E3 +7644.672}
SPL {X  -159.990, Y  +434.697, Z    +0.000, E1   -71.504, E3 +7649.692}
SPL {X  -159.990, Y  +521.523, Z    +0.000, E1   -76.035, E3 +7675.973}
SPL {X  -154.459, Y  +718.205, Z    +0.000, E1   -76.329, E3 +7757.768}
SPL {X  -151.356, Y  +728.349, Z    +0.000, E1   -76.056, E3 +7765.984}
SPL {X  -148.399, Y  +736.287, Z    +0.000, E1   -75.788, E3 +7772.862}
SPL {X  -144.005, Y  +746.209, Z    +0.000, E1   -75.396, E3 +7781.978}
SPL {X  -138.117, Y  +757.250, Z    +0.000, E1   -74.803, E3 +7792.868}
SPL {X  -133.491, Y  +764.686, Z    +0.000, E1   -74.276, E3 +7800.609}
SPL {X  -128.839, Y  +771.354, Z    +0.000, E1   -73.759, E3 +7807.628}
SPL {X  -123.568, Y  +778.125, Z    +0.000, E1   -73.105, E3 +7814.800}
SPL {X  -118.985, Y  +783.455, Z    +0.000, E1   -72.490, E3 +7820.307}
SPL {X   -72.391, Y  +819.176, Z    +0.000, E1   -59.867, E3 +7916.994}
ENDSPLINE

SPLINE
SPL {X   -92.809, Y  +806.820, Z    +0.000, E1   -56.994, E3 +8109.789}
SPL {X  -120.521, Y  +781.721, Z    +0.000, E1   -56.766, E3 +8145.887}
SPL {X  -143.482, Y  +747.279, Z    +0.000, E1   -50.227, E3 +8163.900}
SPL {X  -154.118, Y  +719.449, Z    +0.000, E1   -38.836, E3 +8170.480}
SPL {X  -158.958, Y  +694.646, Z    +0.000, E1   -21.132, E3 +8173.331}
SPL {X  -159.960, Y  +679.609, Z    +0.000, E1    -6.021, E3 +8174.031}
SPL {X  -159.990, Y  +674.508, Z    +0.000, E1    -0.018, E3 +8174.090}
SPL {X  -159.990, Y  +672.787, Z    +0.000, E1    +4.022, E3 +8174.101}
SPL {X  -159.990, Y  +669.267, Z    +0.000, E1   +13.665, E3 +8174.172}
SPL {X  -159.990, Y  +663.438, Z    +0.000, E1   +29.379, E3 +8174.442}
SPL {X  -159.990, Y  +655.264, Z    +0.000, E1   +47.291, E3 +8175.059}
SPL {X  -159.990, Y  +645.368, Z    +0.000, E1   +59.257, E3 +8176.303}
SPL {X  -159.990, Y  +624.023, Z    +0.000, E1   +69.513, E3 +8180.427}
SPL {X  -159.990, Y  +543.075, Z    +0.000, E1   +75.590, E3 +8204.075}
SPL {X  -156.121, Y  +342.530, Z    +0.000, E1   +75.868, E3 +8290.722}
SPL {X  -153.498, Y  +332.386, Z    +0.000, E1   +75.628, E3 +8298.726}
ENDSPLINE

SPLINE
SPL {X  -155.252, Y  +338.851, Z    +0.000, E1   +74.632, E3 +8306.104}
SPL {X  -159.103, Y  +360.678, Z    +0.000, E1   +72.233, E3 +8318.429}
ENDSPLINE

SPLINE
SPL {X  -154.371, Y  +335.471, Z    +0.000, E1   +73.016, E3 +8327.000}
SPL {X  -149.938, Y  +321.685, Z    +0.000, E1   +73.398, E3 +8331.694}
SPL {X  -145.016, Y  +309.920, Z    +0.000, E1   +73.647, E3 +8336.215}
SPL {X  -139.138, Y  +298.522, Z    +0.000, E1   +74.138, E3 +8338.231}
SPL {X  -135.697, Y  +292.747, Z    +0.000, E1   +74.259, E3 +8340.233}
SPL {X  -132.590, Y  +287.964, Z    +0.000, E1   +73.910, E3 +8345.261}
SPL {X  -129.541, Y  +283.606, Z    +0.000, E1   +73.551, E3 +8349.902}
SPL {X  -126.457, Y  +279.493, Z    +0.000, E1   +73.175, E3 +8354.301}
SPL {X  -122.770, Y  +274.912, Z    +0.000, E1   +72.712, E3 +8359.156}
SPL {X  -118.941, Y  +270.496, Z    +0.000, E1   +72.188, E3 +8363.744}
SPL {X   -74.907, Y  +236.129, Z    +0.000, E1   +61.720, E3 +8442.357}
ENDSPLINE

SPLINE
SPL {X   -94.059, Y  +248.080, Z    +0.000, E1   +58.275, E3 +8664.050}
SPL {X  -136.558, Y  +294.141, Z    +0.000, E1   +54.887, E3 +8707.904}
SPL {X  -151.843, Y  +327.098, Z    +0.000, E1   +44.118, E3 +8717.264}
SPL {X  -157.484, Y  +349.293, Z    +0.000, E1   +30.654, E3 +8720.303}
SPL {X  -159.556, Y  +365.719, Z    +0.000, E1   +15.845, E3 +8721.496}
SPL {X  -159.982, Y  +375.924, Z    +0.000, E1    +4.476, E3 +8721.797}
SPL {X  -159.990, Y  +379.531, Z    +0.000, E1    -0.039, E3 +8721.824}
SPL {X  -159.990, Y  +382.420, Z    +0.000, E1    -7.600, E3 +8721.853}
SPL {X  -159.990, Y  +386.504, Z    +0.000, E1   -19.860, E3 +8721.958}
SPL {X  -159.990, Y  +392.530, Z    +0.000, E1   -36.133, E3 +8722.273}
SPL {X  -159.990, Y  +400.492, Z    +0.000, E1   -51.837, E3 +8722.926}
SPL {X  -159.990, Y  +409.662, Z    +0.000, E1   -61.705, E3 +8724.037}
SPL {X  -159.990, Y  +434.697, Z    +0.000, E1   -71.504, E3 +8729.057}
SPL {X  -159.990, Y  +521.523, Z    +0.000, E1   -76.035, E3 +8755.338}
SPL {X  -154.459, Y  +718.205, Z    +0.000, E1   -76.329, E3 +8837.133}
SPL {X  -151.356, Y  +728.349, Z    +0.000, E1   -76.056, E3 +8845.349}
SPL {X  -148.399, Y  +736.287, Z    +0.000, E1   -75.788, E3 +8852.227}
SPL {X  -144.005, Y  +746.209, Z    +0.000, E1   -75.396, E3 +8861.343}
SPL {X  -138.117, Y  +757.250, Z    +0.000, E1   -74.803, E3 +8872.233}
SPL {X  -133.491, Y  +764.686, Z    +0.000, E1   -74.276, E3 +8879.974}
SPL {X  -130.530, Y  +769.013, Z    +0.000, E1   -73.929, E3 +8884.556}
SPL {X  -127.734, Y  +772.837, Z    +0.000, E1   -73.601, E3 +8888.609}
SPL {X  -124.765, Y  +776.652, Z    +0.000, E1   -73.233, E3 +8892.643}
SPL {X  -121.376, Y  +780.734, Z    +0.000, E1   -72.804, E3 +8896.904}
SPL {X  -118.281, Y  +784.233, Z    +0.000, E1   -72.371, E3 +8900.473}
SPL {X   -72.391, Y  +819.176, Z    +0.000, E1   -59.867, E3 +8996.359}
ENDSPLINE

SPLINE
SPL {X   -92.809, Y  +806.820, Z    +0.000, E1   -56.994, E3 +9189.154}
SPL {X  -120.521, Y  +781.721, Z    +0.000, E1   -56.766, E3 +9225.253}
SPL {X  -148.710, Y  +735.509, Z    +0.000, E1   -46.282, E3 +9246.534}
SPL {X  -157.559, Y  +704.285, Z    +0.000, E1   -29.037, E3 +9251.863}
SPL {X  -159.430, Y  +689.871, Z    +0.000, E1   -16.582, E3 +9253.013}
SPL {X  -159.960, Y  +679.609, Z    +0.000, E1    -6.021, E3 +9253.396}
SPL {X  -159.990, Y  +674.508, Z    +0.000, E1    -0.018, E3 +9253.455}
SPL {X  -159.990, Y  +672.787, Z    +0.000, E1    +4.022, E3 +9253.466}
SPL {X  -159.990, Y  +669.267, Z    +0.000, E1   +13.665, E3 +9253.537}
SPL {X  -159.990, Y  +665.069, Z    +0.000, E1   +25.376, E3 +9253.709}
SPL {X  -159.990, Y  +657.821, Z    +0.000, E1   +42.408, E3 +9254.211}
SPL {X  -159.990, Y  +645.368, Z    +0.000, E1   +59.257, E3 +9255.668}
SPL {X  -159.990, Y  +624.023, Z    +0.000, E1   +69.513, E3 +9259.792}
SPL {X  -159.990, Y  +543.075, Z    +0.000, E1   +75.590, E3 +9283.440}
SPL {X  -156.121, Y  +342.530, Z    +0.000, E1   +75.868, E3 +9370.087}
SPL {X  -153.498, Y  +332.386, Z    +0.000, E1   +75.628, E3 +9378.091}
ENDSPLINE

SPLINE
SPL {X  -155.252, Y  +338.851, Z    +0.000, E1   +74.632, E3 +9385.469}
SPL {X  -159.644, Y  +366.989, Z    +0.000, E1   +72.058, E3 +9395.218}
ENDSPLINE

SPLINE
SPL {X  -156.933, Y  +346.374, Z    +0.000, E1   +72.645, E3 +9403.107}
SPL {X  -151.144, Y  +325.039, Z    +0.000, E1   +73.323, E3 +9409.787}
SPL {X  -146.668, Y  +313.584, Z    +0.000, E1   +73.560, E3 +9414.268}
SPL {X  -141.230, Y  +302.327, Z    +0.000, E1   +73.933, E3 +9417.240}
SPL {X  -135.697, Y  +292.747, Z    +0.000, E1   +74.259, E3 +9419.598}
SPL {X  -132.590, Y  +287.964, Z    +0.000, E1   +73.910, E3 +9424.626}
SPL {X  -129.541, Y  +283.606, Z    +0.000, E1   +73.551, E3 +9429.267}
SPL {X  -125.403, Y  +278.147, Z    +0.000, E1   +73.063, E3 +9435.074}
SPL {X  -121.908, Y  +273.889, Z    +0.000, E1   +72.578, E3 +9439.620}
SPL {X  -118.941, Y  +270.496, Z    +0.000, E1   +72.188, E3 +9443.109}
SPL {X   -74.907, Y  +236.129, Z    +0.000, E1   +61.720, E3 +9521.722}
SPL {X   -72.759, Y  +235.012, Z    +0.000, E1   +56.036, E3 +9693.399}
ENDSPLINE

SPLINE
SPL {X  -123.257, Y  +275.497, Z    +0.000, E1   +57.800, E3 +9777.275}
SPL {X  -149.689, Y  +321.019, Z    +0.000, E1   +46.817, E3 +9795.376}
SPL {X  -157.484, Y  +349.293, Z    +0.000, E1   +30.654, E3 +9799.668}
SPL {X  -159.556, Y  +365.719, Z    +0.000, E1   +15.845, E3 +9800.861}
SPL {X  -159.982, Y  +375.924, Z    +0.000, E1    +4.476, E3 +9801.163}
SPL {X  -159.990, Y  +379.531, Z    +0.000, E1    -0.039, E3 +9801.190}
SPL {X  -159.990, Y  +382.420, Z    +0.000, E1    -7.600, E3 +9801.218}
SPL {X  -159.990, Y  +387.978, Z    +0.000, E1   -23.882, E3 +9801.386}
SPL {X  -159.990, Y  +396.850, Z    +0.000, E1   -45.459, E3 +9801.973}
SPL {X  -159.990, Y  +409.662, Z    +0.000, E1   -61.705, E3 +9803.402}
SPL {X  -159.990, Y  +426.583, Z    +0.000, E1   -69.729, E3 +9806.517}
SPL {X  -159.990, Y  +451.842, Z    +0.000, E1   -73.935, E3 +9812.443}
SPL {X  -159.990, Y  +521.523, Z    +0.000, E1   -76.035, E3 +9834.703}
SPL {X  -154.459, Y  +718.205, Z    +0.000, E1   -76.329, E3 +9916.498}
SPL {X  -151.356, Y  +728.349, Z    +0.000, E1   -76.056, E3 +9924.714}
SPL {X  -148.399, Y  +736.287, Z    +0.000, E1   -75.788, E3 +9931.593}
SPL {X  -144.005, Y  +746.209, Z    +0.000, E1   -75.396, E3 +9940.708}
SPL {X  -138.117, Y  +757.250, Z    +0.000, E1   -74.803, E3 +9951.599}
SPL {X  -133.491, Y  +764.686, Z    +0.000, E1   -74.276, E3 +9959.339}
SPL {X  -130.530, Y  +769.013, Z    +0.000, E1   -73.929, E3 +9963.921}
SPL {X  -127.734, Y  +772.837, Z    +0.000, E1   -73.601, E3 +9967.974}
SPL {X  -123.568, Y  +778.125, Z    +0.000, E1   -73.105, E3 +9973.530}
SPL {X  -118.985, Y  +783.455, Z    +0.000, E1   -72.490, E3 +9979.037}
SPL {X   -72.391, Y  +819.176, Z    +0.000, E1   -59.867, E3 +10075.724}
ENDSPLINE

SPLINE
SPL {X  -116.241, Y  +786.431, Z    +0.000, E1   -57.120, E3 +10300.166}
SPL {X  -148.710, Y  +735.509, Z    +0.000, E1   -46.282, E3 +10325.899}
SPL {X  -156.039, Y  +711.834, Z    +0.000, E1   -34.227, E3 +10330.384}
SPL {X  -158.281, Y  +699.823, Z    +0.000, E1   -25.469, E3 +10331.674}
SPL {X  -159.709, Y  +685.986, Z    +0.000, E1   -12.810, E3 +10332.560}
SPL {X  -159.990, Y  +674.648, Z    +0.000, E1    -0.349, E3 +10332.819}
SPL {X  -159.990, Y  +672.787, Z    +0.000, E1    +4.022, E3 +10332.832}
SPL {X  -159.990, Y  +669.267, Z    +0.000, E1   +13.665, E3 +10332.902}
SPL {X  -159.990, Y  +665.069, Z    +0.000, E1   +25.376, E3 +10333.074}
SPL {X  -159.990, Y  +657.821, Z    +0.000, E1   +42.408, E3 +10333.576}
SPL {X  -159.990, Y  +645.368, Z    +0.000, E1   +59.257, E3 +10335.033}
SPL {X  -159.990, Y  +624.023, Z    +0.000, E1   +69.513, E3 +10339.158}
SPL {X  -159.990, Y  +543.075, Z    +0.000, E1   +75.590, E3 +10362.806}
SPL {X  -156.121, Y  +342.530, Z    +0.000, E1   +75.868, E3 +10449.452}
SPL {X  -153.498, Y  +332.386, Z    +0.000, E1   +75.628, E3 +10457.456}
ENDSPLINE

SPLINE
SPL {X  -155.252, Y  +338.851, Z    +0.000, E1   +74.632, E3 +10464.835}
SPL {X  -159.103, Y  +360.678, Z    +0.000, E1   +72.233, E3 +10477.159}
ENDSPLINE

SPLINE
SPL {X  -154.371, Y  +335.471, Z    +0.000, E1   +73.016, E3 +10485.730}
SPL {X  -149.938, Y  +321.685, Z    +0.000, E1   +73.398, E3 +10490.425}
SPL {X  -145.016, Y  +309.920, Z    +0.000, E1   +73.647, E3 +10494.945}
SPL {X  -139.138, Y  +298.522, Z    +0.000, E1   +74.138, E3 +10496.961}
SPL {X  -135.697, Y  +292.747, Z    +0.000, E1   +74.259, E3 +10498.963}
SPL {X  -132.590, Y  +287.964, Z    +0.000, E1   +73.910, E3 +10503.991}
SPL {X  -129.541, Y  +283.606, Z    +0.000, E1   +73.551, E3 +10508.632}
SPL {X  -126.457, Y  +279.493, Z    +0.000, E1   +73.175, E3 +10513.031}
SPL {X  -122.770, Y  +274.912, Z    +0.000, E1   +72.712, E3 +10517.886}
SPL {X  -119.156, Y  +270.736, Z    +0.000, E1   +72.213, E3 +10522.236}
SPL {X  -117.531, Y  +268.949, Z    +0.000, E1   +71.964, E3 +10524.051}
SPL {X   -74.907, Y  +236.129, Z    +0.000, E1   +61.720, E3 +10601.087}
ENDSPLINE

SPLINE
SPL {X   -94.059, Y  +248.080, Z    +0.000, E1   +58.275, E3 +10822.780}
SPL {X  -130.769, Y  +285.325, Z    +0.000, E1   +56.495, E3 +10862.657}
SPL {X  -149.689, Y  +321.019, Z    +0.000, E1   +46.817, E3 +10874.741}
SPL {X  -157.484, Y  +349.293, Z    +0.000, E1   +30.654, E3 +10879.033}
SPL {X  -159.556, Y  +365.719, Z    +0.000, E1   +15.845, E3 +10880.226}
SPL {X  -159.982, Y  +375.924, Z    +0.000, E1    +4.476, E3 +10880.528}
SPL {X  -159.990, Y  +379.531, Z    +0.000, E1    -0.039, E3 +10880.555}
SPL {X  -159.990, Y  +382.420, Z    +0.000, E1    -7.600, E3 +10880.583}
SPL {X  -159.990, Y  +386.504, Z    +0.000, E1   -19.860, E3 +10880.688}
SPL {X  -159.990, Y  +392.530, Z    +0.000, E1   -36.133, E3 +10881.004}
SPL {X  -159.990, Y  +400.492, Z    +0.000, E1   -51.837, E3 +10881.656}
SPL {X  -159.990, Y  +409.662, Z    +0.000, E1   -61.705, E3 +10882.768}
SPL {X  -159.990, Y  +434.697, Z    +0.000, E1   -71.504, E3 +10887.788}
SPL {X  -159.990, Y  +521.523, Z    +0.000, E1   -76.035, E3 +10914.068}
SPL {X  -154.459, Y  +718.205, Z    +0.000, E1   -76.329, E3 +10995.863}
SPL {X  -151.356, Y  +728.349, Z    +0.000, E1   -76.056, E3 +11004.079}
SPL {X  -148.399, Y  +736.287, Z    +0.000, E1   -75.788, E3 +11010.958}
SPL {X  -144.005, Y  +746.209, Z    +0.000, E1   -75.396, E3 +11020.074}
SPL {X  -138.117, Y  +757.250, Z    +0.000, E1   -74.803, E3 +11030.964}
SPL {X  -133.491, Y  +764.686, Z    +0.000, E1   -74.276, E3 +11038.705}
SPL {X  -128.839, Y  +771.354, Z    +0.000, E1   -73.759, E3 +11045.723}
SPL {X  -123.568, Y  +778.125, Z    +0.000, E1   -73.105, E3 +11052.895}
SPL {X  -118.985, Y  +783.455, Z    +0.000, E1   -72.490, E3 +11058.402}
SPL {X   -72.391, Y  +819.176, Z    +0.000, E1   -59.867, E3 +11155.089}
ENDSPLINE

SPLINE
SPL {X   -92.809, Y  +806.820, Z    +0.000, E1   -56.994, E3 +11347.884}
SPL {X  -120.521, Y  +781.721, Z    +0.000, E1   -56.766, E3 +11383.983}
SPL {X  -148.710, Y  +735.509, Z    +0.000, E1   -46.282, E3 +11405.264}
SPL {X  -157.559, Y  +704.285, Z    +0.000, E1   -29.037, E3 +11410.593}
SPL {X  -159.430, Y  +689.871, Z    +0.000, E1   -16.582, E3 +11411.743}
SPL {X  -159.960, Y  +679.609, Z    +0.000, E1    -6.021, E3 +11412.126}
SPL {X  -159.990, Y  +674.508, Z    +0.000, E1    -0.018, E3 +11412.185}
SPL {X  -159.990, Y  +672.787, Z    +0.000, E1    +4.022, E3 +11412.197}
SPL {X  -159.990, Y  +669.267, Z    +0.000, E1   +13.665, E3 +11412.267}
SPL {X  -159.990, Y  +663.438, Z    +0.000, E1   +29.379, E3 +11412.538}
SPL {X  -159.990, Y  +655.264, Z    +0.000, E1   +47.291, E3 +11413.154}
SPL {X  -159.990, Y  +645.368, Z    +0.000, E1   +59.257, E3 +11414.398}
SPL {X  -159.990, Y  +624.023, Z    +0.000, E1   +69.513, E3 +11418.523}
SPL {X  -159.990, Y  +543.075, Z    +0.000, E1   +75.590, E3 +11442.171}
SPL {X  -156.121, Y  +342.530, Z    +0.000, E1   +75.868, E3 +11528.817}
SPL {X  -153.865, Y  +333.657, Z    +0.000, E1   +75.438, E3 +11538.421}
ENDSPLINE

SPLINE
SPL {X  -159.103, Y  +360.678, Z    +0.000, E1   +72.233, E3 +11556.525}
ENDSPLINE

SPLINE
SPL {X  -154.371, Y  +335.471, Z    +0.000, E1   +73.016, E3 +11565.095}
SPL {X  -148.318, Y  +317.512, Z    +0.000, E1   +73.488, E3 +11571.417}
SPL {X  -141.230, Y  +302.327, Z    +0.000, E1   +73.933, E3 +11575.970}
SPL {X  -135.697, Y  +292.747, Z    +0.000, E1   +74.259, E3 +11578.328}
SPL {X  -132.590, Y  +287.964, Z    +0.000, E1   +73.910, E3 +11583.356}
SPL {X  -129.541, Y  +283.606, Z    +0.000, E1   +73.551, E3 +11587.997}
SPL {X  -126.457, Y  +279.493, Z    +0.000, E1   +73.175, E3 +11592.396}
SPL {X  -122.770, Y  +274.912, Z    +0.000, E1   +72.712, E3 +11597.251}
SPL {X  -119.156, Y  +270.736, Z    +0.000, E1   +72.213, E3 +11601.601}
SPL {X  -117.531, Y  +268.949, Z    +0.000, E1   +71.964, E3 +11603.416}
SPL {X   -74.907, Y  +236.129, Z    +0.000, E1   +61.720, E3 +11680.452}
SPL {X   -72.759, Y  +235.012, Z    +0.000, E1   +56.036, E3 +11852.130}
ENDSPLINE

SPLINE
SPL {X  -110.316, Y  +261.624, Z    +0.000, E1   +58.739, E3 +11924.202}
SPL {X  -136.558, Y  +294.141, Z    +0.000, E1   +54.887, E3 +11945.999}
SPL {X  -153.807, Y  +333.452, Z    +0.000, E1   +40.945, E3 +11956.396}
SPL {X  -158.168, Y  +353.421, Z    +0.000, E1   +27.296, E3 +11958.790}
SPL {X  -159.556, Y  +365.719, Z    +0.000, E1   +15.845, E3 +11959.591}
SPL {X  -159.982, Y  +375.924, Z    +0.000, E1    +4.476, E3 +11959.893}
SPL {X  -159.990, Y  +379.800, Z    +0.000, E1    -0.377, E3 +11959.921}
SPL {X  -159.990, Y  +383.422, Z    +0.000, E1   -10.730, E3 +11959.964}
SPL {X  -159.990, Y  +387.978, Z    +0.000, E1   -23.882, E3 +11960.116}
SPL {X  -159.990, Y  +394.494, Z    +0.000, E1   -40.961, E3 +11960.497}
SPL {X  -159.990, Y  +400.492, Z    +0.000, E1   -51.837, E3 +11961.022}
SPL {X  -159.990, Y  +409.662, Z    +0.000, E1   -61.705, E3 +11962.133}
SPL {X  -159.990, Y  +434.697, Z    +0.000, E1   -71.504, E3 +11967.153}
SPL {X  -159.990, Y  +521.523, Z    +0.000, E1   -76.035, E3 +11993.433}
SPL {X  -154.459, Y  +718.205, Z    +0.000, E1   -76.329, E3 +12075.229}
SPL {X  -151.356, Y  +728.349, Z    +0.000, E1   -76.056, E3 +12083.444}
SPL {X  -148.399, Y  +736.287, Z    +0.000, E1   -75.788, E3 +12090.323}
SPL {X  -144.005, Y  +746.209, Z    +0.000, E1   -75.396, E3 +12099.439}
SPL {X  -138.117, Y  +757.250, Z    +0.000, E1   -74.803, E3 +12110.329}
SPL {X  -133.491, Y  +764.686, Z    +0.000, E1   -74.276, E3 +12118.070}
SPL {X  -128.839, Y  +771.354, Z    +0.000, E1   -73.759, E3 +12125.088}
SPL {X  -124.765, Y  +776.652, Z    +0.000, E1   -73.233, E3 +12130.738}
SPL {X  -121.376, Y  +780.734, Z    +0.000, E1   -72.804, E3 +12135.000}
SPL {X  -118.281, Y  +784.233, Z    +0.000, E1   -72.371, E3 +12138.568}
SPL {X   -72.391, Y  +819.176, Z    +0.000, E1   -59.867, E3 +12234.454}
ENDSPLINE

SPLINE
SPL {X  -116.241, Y  +786.431, Z    +0.000, E1   -57.120, E3 +12458.896}
SPL {X  -148.710, Y  +735.509, Z    +0.000, E1   -46.282, E3 +12484.629}
SPL {X  -157.559, Y  +704.285, Z    +0.000, E1   -29.037, E3 +12489.958}
SPL {X  -159.709, Y  +685.986, Z    +0.000, E1   -12.810, E3 +12491.290}
SPL {X  -159.990, Y  +674.648, Z    +0.000, E1    -0.349, E3 +12491.549}
SPL {X  -159.990, Y  +672.787, Z    +0.000, E1    +4.022, E3 +12491.562}
SPL {X  -159.990, Y  +669.267, Z    +0.000, E1   +13.665, E3 +12491.632}
SPL {X  -159.990, Y  +665.069, Z    +0.000, E1   +25.376, E3 +12491.804}
SPL {X  -159.990, Y  +657.821, Z    +0.000, E1   +42.408, E3 +12492.306}
SPL {X  -159.990, Y  +645.368, Z    +0.000, E1   +59.257, E3 +12493.763}
SPL {X  -159.990, Y  +624.023, Z    +0.000, E1   +69.513, E3 +12497.888}
SPL {X  -159.990, Y  +543.075, Z    +0.000, E1   +75.590, E3 +12521.536}
SPL {X  -156.121, Y  +342.530, Z    +0.000, E1   +75.868, E3 +12608.182}
SPL {X  -153.865, Y  +333.657, Z    +0.000, E1   +75.438, E3 +12617.786}
ENDSPLINE

SPLINE
SPL {X  -159.103, Y  +360.678, Z    +0.000, E1   +72.233, E3 +12635.890}
ENDSPLINE

SPLINE
SPL {X  -154.371, Y  +335.471, Z    +0.000, E1   +73.016, E3 +12644.460}
SPL {X  -149.938, Y  +321.685, Z    +0.000, E1   +73.398, E3 +12649.155}
SPL {X  -145.016, Y  +309.920, Z    +0.000, E1   +73.647, E3 +12653.676}
SPL {X  -139.138, Y  +298.522, Z    +0.000, E1   +74.138, E3 +12655.692}
SPL {X  -135.697, Y  +292.747, Z    +0.000, E1   +74.259, E3 +12657.693}
SPL {X  -132.590, Y  +287.964, Z    +0.000, E1   +73.910, E3 +12662.722}
SPL {X  -129.541, Y  +283.606, Z    +0.000, E1   +73.551, E3 +12667.362}
SPL {X  -126.457, Y  +279.493, Z    +0.000, E1   +73.175, E3 +12671.761}
SPL {X  -122.770, Y  +274.912, Z    +0.000, E1   +72.712, E3 +12676.616}
SPL {X  -118.941, Y  +270.496, Z    +0.000, E1   +72.188, E3 +12681.204}
SPL {X   -74.907, Y  +236.129, Z    +0.000, E1   +61.720, E3 +12759.817}
ENDSPLINE

SPLINE
SPL {X   -94.059, Y  +248.080, Z    +0.000, E1   +58.275, E3 +12981.510}
SPL {X  -130.769, Y  +285.325, Z    +0.000, E1   +56.495, E3 +13021.387}
SPL {X  -149.689, Y  +321.019, Z    +0.000, E1   +46.817, E3 +13033.471}
SPL {X  -155.950, Y  +341.772, Z    +0.000, E1   +35.915, E3 +13036.970}
SPL {X  -158.168, Y  +353.421, Z    +0.000, E1   +27.296, E3 +13038.155}
SPL {X  -159.556, Y  +365.719, Z    +0.000, E1   +15.845, E3 +13038.956}
SPL {X  -159.982, Y  +375.924, Z    +0.000, E1    +4.476, E3 +13039.258}
SPL {X  -159.990, Y  +379.800, Z    +0.000, E1    -0.377, E3 +13039.286}
SPL {X  -159.990, Y  +385.115, Z    +0.000, E1   -15.358, E3 +13039.378}
SPL {X  -159.990, Y  +392.530, Z    +0.000, E1   -36.133, E3 +13039.734}
SPL {X  -159.990, Y  +400.492, Z    +0.000, E1   -51.837, E3 +13040.387}
SPL {X  -159.990, Y  +409.662, Z    +0.000, E1   -61.705, E3 +13041.498}
SPL {X  -159.990, Y  +434.697, Z    +0.000, E1   -71.504, E3 +13046.518}
SPL {X  -159.990, Y  +521.523, Z    +0.000, E1   -76.035, E3 +13072.798}
SPL {X  -154.459, Y  +718.205, Z    +0.000, E1   -76.329, E3 +13154.594}
SPL {X  -151.356, Y  +728.349, Z    +0.000, E1   -76.056, E3 +13162.809}
SPL {X  -147.124, Y  +739.360, Z    +0.000, E1   -75.690, E3 +13172.405}
SPL {X  -142.861, Y  +748.524, Z    +0.000, E1   -75.261, E3 +13181.090}
SPL {X  -138.117, Y  +757.250, Z    +0.000, E1   -74.803, E3 +13189.694}
SPL {X  -133.491, Y  +764.686, Z    +0.000, E1   -74.276, E3 +13197.435}
SPL {X  -130.530, Y  +769.013, Z    +0.000, E1   -73.929, E3 +13202.017}
SPL {X  -127.734, Y  +772.837, Z    +0.000, E1   -73.601, E3 +13206.069}
SPL {X  -124.765, Y  +776.652, Z    +0.000, E1   -73.233, E3 +13210.103}
SPL {X  -121.376, Y  +780.734, Z    +0.000, E1   -72.804, E3 +13214.365}
SPL {X  -118.281, Y  +784.233, Z    +0.000, E1   -72.371, E3 +13217.933}
SPL {X   -72.391, Y  +819.176, Z    +0.000, E1   -59.867, E3 +13313.819}
ENDSPLINE

SPLINE
SPL {X  -116.241, Y  +786.431, Z    +0.000, E1   -57.120, E3 +13538.261}
SPL {X  -148.710, Y  +735.509, Z    +0.000, E1   -46.282, E3 +13563.994}
SPL {X  -156.039, Y  +711.834, Z    +0.000, E1   -34.227, E3 +13568.479}
SPL {X  -158.958, Y  +694.646, Z    +0.000, E1   -21.132, E3 +13570.156}
SPL {X  -159.960, Y  +679.609, Z    +0.000, E1    -6.021, E3 +13570.856}
SPL {X  -159.990, Y  +674.508, Z    +0.000, E1    -0.018, E3 +13570.915}
SPL {X  -159.990, Y  +672.787, Z    +0.000, E1    +4.022, E3 +13570.927}
SPL {X  -159.990, Y  +669.267, Z    +0.000, E1   +13.665, E3 +13570.997}
SPL {X  -159.990, Y  +663.438, Z    +0.000, E1   +29.379, E3 +13571.268}
SPL {X  -159.990, Y  +655.264, Z    +0.000, E1   +47.291, E3 +13571.885}
SPL {X  -159.990, Y  +645.368, Z    +0.000, E1   +59.257, E3 +13573.128}
SPL {X  -159.990, Y  +624.023, Z    +0.000, E1   +69.513, E3 +13577.253}
SPL {X  -159.990, Y  +543.075, Z    +0.000, E1   +75.590, E3 +13600.901}
SPL {X  -156.121, Y  +342.530, Z    +0.000, E1   +75.868, E3 +13687.547}
SPL {X  -153.865, Y  +333.657, Z    +0.000, E1   +75.438, E3 +13697.151}
ENDSPLINE

SPLINE
SPL {X  -159.103, Y  +360.678, Z    +0.000, E1   +72.233, E3 +13715.255}
ENDSPLINE

SPLINE
SPL {X  -154.371, Y  +335.471, Z    +0.000, E1   +73.016, E3 +13723.825}
SPL {X  -149.938, Y  +321.685, Z    +0.000, E1   +73.398, E3 +13728.520}
SPL {X  -145.016, Y  +309.920, Z    +0.000, E1   +73.647, E3 +13733.041}
SPL {X  -139.138, Y  +298.522, Z    +0.000, E1   +74.138, E3 +13735.057}
SPL {X  -135.697, Y  +292.747, Z    +0.000, E1   +74.259, E3 +13737.059}
SPL {X  -132.590, Y  +287.964, Z    +0.000, E1   +73.910, E3 +13742.087}
SPL {X  -129.541, Y  +283.606, Z    +0.000, E1   +73.551, E3 +13746.727}
SPL {X  -125.403, Y  +278.147, Z    +0.000, E1   +73.063, E3 +13752.534}
SPL {X  -121.908, Y  +273.889, Z    +0.000, E1   +72.578, E3 +13757.081}
SPL {X  -118.941, Y  +270.496, Z    +0.000, E1   +72.188, E3 +13760.569}
SPL {X   -74.907, Y  +236.129, Z    +0.000, E1   +61.720, E3 +13839.182}
SPL {X   -72.759, Y  +235.012, Z    +0.000, E1   +56.036, E3 +14010.860}
ENDSPLINE

SPLINE
SPL {X  -123.257, Y  +275.497, Z    +0.000, E1   +57.800, E3 +14094.736}
SPL {X  -149.689, Y  +321.019, Z    +0.000, E1   +46.817, E3 +14112.836}
SPL {X  -155.950, Y  +341.772, Z    +0.000, E1   +35.915, E3 +14116.335}
SPL {X  -158.168, Y  +353.421, Z    +0.000, E1   +27.296, E3 +14117.520}
SPL {X  -159.556, Y  +365.719, Z    +0.000, E1   +15.845, E3 +14118.321}
SPL {X  -159.982, Y  +375.924, Z    +0.000, E1    +4.476, E3 +14118.623}
SPL {X  -159.990, Y  +379.800, Z    +0.000, E1    -0.377, E3 +14118.651}
SPL {X  -159.990, Y  +385.115, Z    +0.000, E1   -15.358, E3 +14118.743}
SPL {X  -159.990, Y  +392.530, Z    +0.000, E1   -36.133, E3 +14119.099}
SPL {X  -159.990, Y  +400.492, Z    +0.000, E1   -51.837, E3 +14119.752}
SPL {X  -159.990, Y  +409.662, Z    +0.000, E1   -61.705, E3 +14120.863}
SPL {X  -159.990, Y  +434.697, Z    +0.000, E1   -71.504, E3 +14125.883}
SPL {X  -159.990, Y  +521.523, Z    +0.000, E1   -76.035, E3 +14152.163}
SPL {X  -154.459, Y  +718.205, Z    +0.000, E1   -76.329, E3 +14233.959}
SPL {X  -151.356, Y  +728.349, Z    +0.000, E1   -76.056, E3 +14242.174}
SPL {X  -148.399, Y  +736.287, Z    +0.000, E1   -75.788, E3 +14249.053}
SPL {X  -144.005, Y  +746.209, Z    +0.000, E1   -75.396, E3 +14258.169}
SPL {X  -138.117, Y  +757.250, Z    +0.000, E1   -74.803, E3 +14269.059}
SPL {X  -133.491, Y  +764.686, Z    +0.000, E1   -74.276, E3 +14276.800}
SPL {X  -128.839, Y  +771.354, Z    +0.000, E1   -73.759, E3 +14283.819}
SPL {X  -123.568, Y  +778.125, Z    +0.000, E1   -73.105, E3 +14290.990}
SPL {X  -118.985, Y  +783.455, Z    +0.000, E1   -72.490, E3 +14296.498}
SPL {X   -72.391, Y  +819.176, Z    +0.000, E1   -59.867, E3 +14393.184}
ENDSPLINE

SPLINE
SPL {X   -92.809, Y  +806.820, Z    +0.000, E1   -56.994, E3 +14585.979}
SPL {X  -120.521, Y  +781.721, Z    +0.000, E1   -56.766, E3 +14622.078}
SPL {X  -143.482, Y  +747.279, Z    +0.000, E1   -50.227, E3 +14640.091}
SPL {X  -154.118, Y  +719.449, Z    +0.000, E1   -38.836, E3 +14646.670}
SPL {X  -158.958, Y  +694.646, Z    +0.000, E1   -21.132, E3 +14649.521}
SPL {X  -159.960, Y  +679.609, Z    +0.000, E1    -6.021, E3 +14650.221}
SPL {X  -159.990, Y  +674.508, Z    +0.000, E1    -0.018, E3 +14650.280}
SPL {X  -159.990, Y  +672.787, Z    +0.000, E1    +4.022, E3 +14650.292}
SPL {X  -159.990, Y  +669.267, Z    +0.000, E1   +13.665, E3 +14650.362}
SPL {X  -159.990, Y  +663.438, Z    +0.000, E1   +29.379, E3 +14650.633}
SPL {X  -159.990, Y  +655.264, Z    +0.000, E1   +47.291, E3 +14651.250}
SPL {X  -159.990, Y  +645.368, Z    +0.000, E1   +59.257, E3 +14652.493}
SPL {X  -159.990, Y  +624.023, Z    +0.000, E1   +69.513, E3 +14656.618}
SPL {X  -159.990, Y  +543.075, Z    +0.000, E1   +75.590, E3 +14680.266}
SPL {X  -156.121, Y  +342.530, Z    +0.000, E1   +75.868, E3 +14766.912}
SPL {X  -153.498, Y  +332.386, Z    +0.000, E1   +75.628, E3 +14774.917}
ENDSPLINE

SPLINE
SPL {X  -155.252, Y  +338.851, Z    +0.000, E1   +74.632, E3 +14782.295}
SPL {X  -159.103, Y  +360.678, Z    +0.000, E1   +72.233, E3 +14794.620}
ENDSPLINE

SPLINE
SPL {X  -154.371, Y  +335.471, Z    +0.000, E1   +73.016, E3 +14803.191}
SPL {X  -149.938, Y  +321.685, Z    +0.000, E1   +73.398, E3 +14807.885}
SPL {X  -145.016, Y  +309.920, Z    +0.000, E1   +73.647, E3 +14812.406}
SPL {X  -139.138, Y  +298.522, Z    +0.000, E1   +74.138, E3 +14814.422}
SPL {X  -135.697, Y  +292.747, Z    +0.000, E1   +74.259, E3 +14816.424}
SPL {X  -132.590, Y  +287.964, Z    +0.000, E1   +73.910, E3 +14821.452}
SPL {X  -129.541, Y  +283.606, Z    +0.000, E1   +73.551, E3 +14826.092}
SPL {X  -126.457, Y  +279.493, Z    +0.000, E1   +73.175, E3 +14830.491}
SPL {X  -122.770, Y  +274.912, Z    +0.000, E1   +72.712, E3 +14835.347}
SPL {X  -118.941, Y  +270.496, Z    +0.000, E1   +72.188, E3 +14839.934}
SPL {X   -74.907, Y  +236.129, Z    +0.000, E1   +61.720, E3 +14918.547}
ENDSPLINE

SPLINE
SPL {X   -94.059, Y  +248.080, Z    +0.000, E1   +58.275, E3 +15140.240}
SPL {X  -136.558, Y  +294.141, Z    +0.000, E1   +54.887, E3 +15184.095}
SPL {X  -151.843, Y  +327.098, Z    +0.000, E1   +44.118, E3 +15193.454}
SPL {X  -157.484, Y  +349.293, Z    +0.000, E1   +30.654, E3 +15196.494}
SPL {X  -159.556, Y  +365.719, Z    +0.000, E1   +15.845, E3 +15197.686}
SPL {X  -159.982, Y  +375.924, Z    +0.000, E1    +4.476, E3 +15197.988}
SPL {X  -159.990, Y  +379.531, Z    +0.000, E1    -0.039, E3 +15198.015}
SPL {X  -159.990, Y  +382.420, Z    +0.000, E1    -7.600, E3 +15198.043}
SPL {X  -159.990, Y  +386.504, Z    +0.000, E1   -19.860, E3 +15198.149}
SPL {X  -159.990, Y  +392.530, Z    +0.000, E1   -36.133, E3 +15198.464}
SPL {X  -159.990, Y  +400.492, Z    +0.000, E1   -51.837, E3 +15199.117}
SPL {X  -159.990, Y  +409.662, Z    +0.000, E1   -61.705, E3 +15200.228}
SPL {X  -159.990, Y  +434.697, Z    +0.000, E1   -71.504, E3 +15205.248}
SPL {X  -159.990, Y  +521.523, Z    +0.000, E1   -76.035, E3 +15231.528}
SPL {X  -154.459, Y  +718.205, Z    +0.000, E1   -76.329, E3 +15313.324}
SPL {X  -151.356, Y  +728.349, Z    +0.000, E1   -76.056, E3 +15321.539}
SPL {X  -148.399, Y  +736.287, Z    +0.000, E1   -75.788, E3 +15328.418}
SPL {X  -144.005, Y  +746.209, Z    +0.000, E1   -75.396, E3 +15337.534}
SPL {X  -138.117, Y  +757.250, Z    +0.000, E1   -74.803, E3 +15348.424}
SPL {X  -133.491, Y  +764.686, Z    +0.000, E1   -74.276, E3 +15356.165}
SPL {X  -128.839, Y  +771.354, Z    +0.000, E1   -73.759, E3 +15363.184}
SPL {X  -123.568, Y  +778.125, Z    +0.000, E1   -73.105, E3 +15370.355}
SPL {X  -118.985, Y  +783.455, Z    +0.000, E1   -72.490, E3 +15375.863}
SPL {X   -72.391, Y  +819.176, Z    +0.000, E1   -59.867, E3 +15472.549}
ENDSPLINE

SPLINE
SPL {X   -92.809, Y  +806.820, Z    +0.000, E1   -56.994, E3 +15665.344}
SPL {X  -120.521, Y  +781.721, Z    +0.000, E1   -56.766, E3 +15701.443}
SPL {X  -148.710, Y  +735.509, Z    +0.000, E1   -46.282, E3 +15722.724}
SPL {X  -157.559, Y  +704.285, Z    +0.000, E1   -29.037, E3 +15728.053}
SPL {X  -159.430, Y  +689.871, Z    +0.000, E1   -16.582, E3 +15729.203}
SPL {X  -159.960, Y  +679.609, Z    +0.000, E1    -6.021, E3 +15729.587}
SPL {X  -159.990, Y  +674.508, Z    +0.000, E1    -0.018, E3 +15729.645}
SPL {X  -159.990, Y  +672.787, Z    +0.000, E1    +4.022, E3 +15729.657}
SPL {X  -159.990, Y  +669.267, Z    +0.000, E1   +13.665, E3 +15729.727}
SPL {X  -159.990, Y  +663.438, Z    +0.000, E1   +29.379, E3 +15729.998}
SPL {X  -159.990, Y  +655.264, Z    +0.000, E1   +47.291, E3 +15730.615}
SPL {X  -159.990, Y  +645.368, Z    +0.000, E1   +59.257, E3 +15731.858}
SPL {X  -159.990, Y  +624.023, Z    +0.000, E1   +69.513, E3 +15735.983}
SPL {X  -159.990, Y  +543.075, Z    +0.000, E1   +75.590, E3 +15759.631}
SPL {X  -156.121, Y  +342.530, Z    +0.000, E1   +75.868, E3 +15846.277}
SPL {X  -153.865, Y  +333.657, Z    +0.000, E1   +75.438, E3 +15855.881}
ENDSPLINE

SPLINE
SPL {X  -159.644, Y  +366.989, Z    +0.000, E1   +72.058, E3 +15871.408}
ENDSPLINE

SPLINE
SPL {X  -156.933, Y  +346.374, Z    +0.000, E1   +72.645, E3 +15879.297}
SPL {X  -151.144, Y  +325.039, Z    +0.000, E1   +73.323, E3 +15885.977}
SPL {X  -145.016, Y  +309.920, Z    +0.000, E1   +73.647, E3 +15891.771}
SPL {X  -136.944, Y  +294.777, Z    +0.000, E1   +74.219, E3 +15895.073}
SPL {X  -132.590, Y  +287.964, Z    +0.000, E1   +73.910, E3 +15900.817}
SPL {X  -129.541, Y  +283.606, Z    +0.000, E1   +73.551, E3 +15905.457}
SPL {X  -125.403, Y  +278.147, Z    +0.000, E1   +73.063, E3 +15911.264}
SPL {X  -121.908, Y  +273.889, Z    +0.000, E1   +72.578, E3 +15915.811}
SPL {X  -118.941, Y  +270.496, Z    +0.000, E1   +72.188, E3 +15919.299}
SPL {X   -74.907, Y  +236.129, Z    +0.000, E1   +61.720, E3 +15997.912}
ENDSPLINE

SPLINE
SPL {X   -94.059, Y  +248.080, Z    +0.000, E1   +58.275, E3 +16219.605}
SPL {X  -136.558, Y  +294.141, Z    +0.000, E1   +54.887, E3 +16263.460}
SPL {X  -151.843, Y  +327.098, Z    +0.000, E1   +44.118, E3 +16272.819}
SPL {X  -157.484, Y  +349.293, Z    +0.000, E1   +30.654, E3 +16275.859}
SPL {X  -159.556, Y  +365.719, Z    +0.000, E1   +15.845, E3 +16277.051}
SPL {X  -159.982, Y  +375.924, Z    +0.000, E1    +4.476, E3 +16277.353}
SPL {X  -159.990, Y  +379.531, Z    +0.000, E1    -0.039, E3 +16277.380}
SPL {X  -159.990, Y  +382.420, Z    +0.000, E1    -7.600, E3 +16277.408}
SPL {X  -159.990, Y  +386.504, Z    +0.000, E1   -19.860, E3 +16277.514}
SPL {X  -159.990, Y  +392.530, Z    +0.000, E1   -36.133, E3 +16277.829}
SPL {X  -159.990, Y  +400.492, Z    +0.000, E1   -51.837, E3 +16278.482}
SPL {X  -159.990, Y  +409.662, Z    +0.000, E1   -61.705, E3 +16279.593}
SPL {X  -159.990, Y  +434.697, Z    +0.000, E1   -71.504, E3 +16284.613}
SPL {X  -159.990, Y  +521.523, Z    +0.000, E1   -76.035, E3 +16310.894}
SPL {X  -154.459, Y  +718.205, Z    +0.000, E1   -76.329, E3 +16392.689}
SPL {X  -151.356, Y  +728.349, Z    +0.000, E1   -76.056, E3 +16400.904}
SPL {X  -147.124, Y  +739.360, Z    +0.000, E1   -75.690, E3 +16410.501}
SPL {X  -142.861, Y  +748.524, Z    +0.000, E1   -75.261, E3 +16419.186}
SPL {X  -139.796, Y  +754.307, Z    +0.000, E1   -74.951, E3 +16424.874}
SPL {X  -136.850, Y  +759.378, Z    +0.000, E1   -74.643, E3 +16430.018}
SPL {X  -133.491, Y  +764.686, Z    +0.000, E1   -74.276, E3 +16435.530}
SPL {X  -128.839, Y  +771.354, Z    +0.000, E1   -73.759, E3 +16442.549}
SPL {X  -124.765, Y  +776.652, Z    +0.000, E1   -73.233, E3 +16448.199}
SPL {X  -121.376, Y  +780.734, Z    +0.000, E1   -72.804, E3 +16452.460}
SPL {X  -118.281, Y  +784.233, Z    +0.000, E1   -72.371, E3 +16456.028}
SPL {X   -72.391, Y  +819.176, Z    +0.000, E1   -59.867, E3 +16551.914}
ENDSPLINE

SPLINE
SPL {X  -116.241, Y  +786.431, Z    +0.000, E1   -57.120, E3 +16776.356}
SPL {X  -148.710, Y  +735.509, Z    +0.000, E1   -46.282, E3 +16802.089}
SPL {X  -156.039, Y  +711.834, Z    +0.000, E1   -34.227, E3 +16806.575}
SPL {X  -158.281, Y  +699.823, Z    +0.000, E1   -25.469, E3 +16807.865}
SPL {X  -159.709, Y  +685.986, Z    +0.000, E1   -12.810, E3 +16808.750}
SPL {X  -159.990, Y  +674.648, Z    +0.000, E1    -0.349, E3 +16809.010}
SPL {X  -159.990, Y  +672.787, Z    +0.000, E1    +4.022, E3 +16809.022}
SPL {X  -159.990, Y  +669.267, Z    +0.000, E1   +13.665, E3 +16809.092}
SPL {X  -159.990, Y  +665.069, Z    +0.000, E1   +25.376, E3 +16809.264}
SPL {X  -159.990, Y  +657.821, Z    +0.000, E1   +42.408, E3 +16809.766}
SPL {X  -159.990, Y  +645.368, Z    +0.000, E1   +59.257, E3 +16811.223}
SPL {X  -159.990, Y  +624.023, Z    +0.000, E1   +69.513, E3 +16815.348}
SPL {X  -159.990, Y  +543.075, Z    +0.000, E1   +75.590, E3 +16838.996}
SPL {X  -156.121, Y  +342.530, Z    +0.000, E1   +75.868, E3 +16925.642}
SPL {X  -153.498, Y  +332.386, Z    +0.000, E1   +75.628, E3 +16933.647}
ENDSPLINE

SPLINE
SPL {X  -155.252, Y  +338.851, Z    +0.000, E1   +74.632, E3 +16941.025}
SPL {X  -159.103, Y  +360.678, Z    +0.000, E1   +72.233, E3 +16953.350}
ENDSPLINE

SPLINE
SPL {X  -154.371, Y  +335.471, Z    +0.000, E1   +73.016, E3 +16961.921}
SPL {X  -149.938, Y  +321.685, Z    +0.000, E1   +73.398, E3 +16966.615}
SPL {X  -145.016, Y  +309.920, Z    +0.000, E1   +73.647, E3 +16971.136}
SPL {X  -139.138, Y  +298.522, Z    +0.000, E1   +74.138, E3 +16973.152}
SPL {X  -135.697, Y  +292.747, Z    +0.000, E1   +74.259, E3 +16975.154}
SPL {X  -132.590, Y  +287.964, Z    +0.000, E1   +73.910, E3 +16980.182}
SPL {X  -129.541, Y  +283.606, Z    +0.000, E1   +73.551, E3 +16984.822}
SPL {X  -126.457, Y  +279.493, Z    +0.000, E1   +73.175, E3 +16989.221}
SPL {X  -122.770, Y  +274.912, Z    +0.000, E1   +72.712, E3 +16994.077}
SPL {X  -119.156, Y  +270.736, Z    +0.000, E1   +72.213, E3 +16998.426}
SPL {X  -117.531, Y  +268.949, Z    +0.000, E1   +71.964, E3 +17000.242}
SPL {X   -74.907, Y  +236.129, Z    +0.000, E1   +61.720, E3 +17077.277}
ENDSPLINE

SPLINE
SPL {X   -94.059, Y  +248.080, Z    +0.000, E1   +58.275, E3 +17298.970}
SPL {X  -130.769, Y  +285.325, Z    +0.000, E1   +56.495, E3 +17338.847}
SPL {X  -149.689, Y  +321.019, Z    +0.000, E1   +46.817, E3 +17350.932}
SPL {X  -157.484, Y  +349.293, Z    +0.000, E1   +30.654, E3 +17355.224}
SPL {X  -159.556, Y  +365.719, Z    +0.000, E1   +15.845, E3 +17356.416}
SPL {X  -159.982, Y  +375.924, Z    +0.000, E1    +4.476, E3 +17356.718}
SPL {X  -159.990, Y  +379.531, Z    +0.000, E1    -0.039, E3 +17356.745}
SPL {X  -159.990, Y  +382.420, Z    +0.000, E1    -7.600, E3 +17356.773}
SPL {X  -159.990, Y  +386.504, Z    +0.000, E1   -19.860, E3 +17356.879}
SPL {X  -159.990, Y  +392.530, Z    +0.000, E1   -36.133, E3 +17357.194}
SPL {X  -159.990, Y  +400.492, Z    +0.000, E1   -51.837, E3 +17357.847}
SPL {X  -159.990, Y  +409.662, Z    +0.000, E1   -61.705, E3 +17358.958}
SPL {X  -159.990, Y  +434.697, Z    +0.000, E1   -71.504, E3 +17363.978}
SPL {X  -159.990, Y  +521.523, Z    +0.000, E1   -76.035, E3 +17390.259}
SPL {X  -154.459, Y  +718.205, Z    +0.000, E1   -76.329, E3 +17472.054}
SPL {X  -151.356, Y  +728.349, Z    +0.000, E1   -76.056, E3 +17480.270}
SPL {X  -148.399, Y  +736.287, Z    +0.000, E1   -75.788, E3 +17487.148}
SPL {X  -144.005, Y  +746.209, Z    +0.000, E1   -75.396, E3 +17496.264}
SPL {X  -138.117, Y  +757.250, Z    +0.000, E1   -74.803, E3 +17507.154}
SPL {X  -133.491, Y  +764.686, Z    +0.000, E1   -74.276, E3 +17514.895}
SPL {X  -128.839, Y  +771.354, Z    +0.000, E1   -73.759, E3 +17521.914}
SPL {X  -123.568, Y  +778.125, Z    +0.000, E1   -73.105, E3 +17529.085}
SPL {X  -118.985, Y  +783.455, Z    +0.000, E1   -72.490, E3 +17534.593}
SPL {X   -72.391, Y  +819.176, Z    +0.000, E1   -59.867, E3 +17631.279}
ENDSPLINE

SPLINE
SPL {X   -92.809, Y  +806.820, Z    +0.000, E1   -56.994, E3 +17824.074}
SPL {X  -120.521, Y  +781.721, Z    +0.000, E1   -56.766, E3 +17860.173}
SPL {X  -148.710, Y  +735.509, Z    +0.000, E1   -46.282, E3 +17881.454}
SPL {X  -157.559, Y  +704.285, Z    +0.000, E1   -29.037, E3 +17886.783}
SPL {X  -159.430, Y  +689.871, Z    +0.000, E1   -16.582, E3 +17887.934}
SPL {X  -159.960, Y  +679.609, Z    +0.000, E1    -6.021, E3 +17888.317}
SPL {X  -159.990, Y  +674.508, Z    +0.000, E1    -0.018, E3 +17888.375}
SPL {X  -159.990, Y  +672.787, Z    +0.000, E1    +4.022, E3 +17888.387}
SPL {X  -159.990, Y  +669.267, Z    +0.000, E1   +13.665, E3 +17888.457}
SPL {X  -159.990, Y  +663.438, Z    +0.000, E1   +29.379, E3 +17888.728}
SPL {X  -159.990, Y  +655.264, Z    +0.000, E1   +47.291, E3 +17889.345}
SPL {X  -159.990, Y  +645.368, Z    +0.000, E1   +59.257, E3 +17890.588}
SPL {X  -159.990, Y  +624.023, Z    +0.000, E1   +69.513, E3 +17894.713}
SPL {X  -159.990, Y  +543.075, Z    +0.000, E1   +75.590, E3 +17918.361}
SPL {X  -156.121, Y  +342.530, Z    +0.000, E1   +75.868, E3 +18005.007}
SPL {X  -153.865, Y  +333.657, Z    +0.000, E1   +75.438, E3 +18014.611}
ENDSPLINE

SPLINE
SPL {X  -159.103, Y  +360.678, Z    +0.000, E1   +72.233, E3 +18032.715}
ENDSPLINE

SPLINE
SPL {X  -154.371, Y  +335.471, Z    +0.000, E1   +73.016, E3 +18041.286}
SPL {X  -148.318, Y  +317.512, Z    +0.000, E1   +73.488, E3 +18047.607}
SPL {X  -141.230, Y  +302.327, Z    +0.000, E1   +73.933, E3 +18052.160}
SPL {X  -135.697, Y  +292.747, Z    +0.000, E1   +74.259, E3 +18054.519}
SPL {X  -132.590, Y  +287.964, Z    +0.000, E1   +73.910, E3 +18059.547}
SPL {X  -129.541, Y  +283.606, Z    +0.000, E1   +73.551, E3 +18064.188}
SPL {X  -126.457, Y  +279.493, Z    +0.000, E1   +73.175, E3 +18068.587}
SPL {X  -122.770, Y  +274.912, Z    +0.000, E1   +72.712, E3 +18073.442}
SPL {X  -119.156, Y  +270.736, Z    +0.000, E1   +72.213, E3 +18077.791}
SPL {X  -117.531, Y  +268.949, Z    +0.000, E1   +71.964, E3 +18079.607}
SPL {X   -74.907, Y  +236.129, Z    +0.000, E1   +61.720, E3 +18156.643}
SPL {X   -72.759, Y  +235.012, Z    +0.000, E1   +56.036, E3 +18328.320}
ENDSPLINE

SPLINE
SPL {X  -110.316, Y  +261.624, Z    +0.000, E1   +58.739, E3 +18400.393}
SPL {X  -136.558, Y  +294.141, Z    +0.000, E1   +54.887, E3 +18422.190}
SPL {X  -153.807, Y  +333.452, Z    +0.000, E1   +40.945, E3 +18432.587}
SPL {X  -158.168, Y  +353.421, Z    +0.000, E1   +27.296, E3 +18434.980}
SPL {X  -159.556, Y  +365.719, Z    +0.000, E1   +15.845, E3 +18435.782}
SPL {X  -159.982, Y  +375.924, Z    +0.000, E1    +4.476, E3 +18436.083}
SPL {X  -159.990, Y  +379.800, Z    +0.000, E1    -0.377, E3 +18436.112}
SPL {X  -159.990, Y  +383.422, Z    +0.000, E1   -10.730, E3 +18436.155}
SPL {X  -159.990, Y  +387.978, Z    +0.000, E1   -23.882, E3 +18436.307}
SPL {X  -159.990, Y  +394.494, Z    +0.000, E1   -40.961, E3 +18436.688}
SPL {X  -159.990, Y  +400.492, Z    +0.000, E1   -51.837, E3 +18437.212}
SPL {X  -159.990, Y  +409.662, Z    +0.000, E1   -61.705, E3 +18438.323}
SPL {X  -159.990, Y  +434.697, Z    +0.000, E1   -71.504, E3 +18443.343}
SPL {X  -159.990, Y  +521.523, Z    +0.000, E1   -76.035, E3 +18469.624}
SPL {X  -154.459, Y  +718.205, Z    +0.000, E1   -76.329, E3 +18551.419}
SPL {X  -151.356, Y  +728.349, Z    +0.000, E1   -76.056, E3 +18559.635}
SPL {X  -147.124, Y  +739.360, Z    +0.000, E1   -75.690, E3 +18569.231}
SPL {X  -142.861, Y  +748.524, Z    +0.000, E1   -75.261, E3 +18577.916}
SPL {X  -139.796, Y  +754.307, Z    +0.000, E1   -74.951, E3 +18583.604}
SPL {X  -136.850, Y  +759.378, Z    +0.000, E1   -74.643, E3 +18588.748}
SPL {X  -133.491, Y  +764.686, Z    +0.000, E1   -74.276, E3 +18594.260}
SPL {X  -128.839, Y  +771.354, Z    +0.000, E1   -73.759, E3 +18601.279}
SPL {X  -124.765, Y  +776.652, Z    +0.000, E1   -73.233, E3 +18606.929}
SPL {X  -121.376, Y  +780.734, Z    +0.000, E1   -72.804, E3 +18611.190}
SPL {X  -118.281, Y  +784.233, Z    +0.000, E1   -72.371, E3 +18614.759}
SPL {X   -72.391, Y  +819.176, Z    +0.000, E1   -59.867, E3 +18710.644}
ENDSPLINE

SPLINE
SPL {X  -116.241, Y  +786.431, Z    +0.000, E1   -57.120, E3 +18935.087}
SPL {X  -143.482, Y  +747.279, Z    +0.000, E1   -50.227, E3 +18957.551}
SPL {X  -154.118, Y  +719.449, Z    +0.000, E1   -38.836, E3 +18964.130}
SPL {X  -158.958, Y  +694.646, Z    +0.000, E1   -21.132, E3 +18966.982}
SPL {X  -159.960, Y  +679.609, Z    +0.000, E1    -6.021, E3 +18967.682}
SPL {X  -159.990, Y  +674.508, Z    +0.000, E1    -0.018, E3 +18967.740}
SPL {X  -159.990, Y  +672.787, Z    +0.000, E1    +4.022, E3 +18967.752}
SPL {X  -159.990, Y  +669.267, Z    +0.000, E1   +13.665, E3 +18967.822}
SPL {X  -159.990, Y  +665.069, Z    +0.000, E1   +25.376, E3 +18967.994}
SPL {X  -159.990, Y  +657.821, Z    +0.000, E1   +42.408, E3 +18968.497}
SPL {X  -159.990, Y  +645.368, Z    +0.000, E1   +59.257, E3 +18969.953}
SPL {X  -159.990, Y  +624.023, Z    +0.000, E1   +69.513, E3 +18974.078}
SPL {X  -159.990, Y  +543.075, Z    +0.000, E1   +75.590, E3 +18997.726}
SPL {X  -156.121, Y  +342.530, Z    +0.000, E1   +75.868, E3 +19084.372}
SPL {X  -153.865, Y  +333.657, Z    +0.000, E1   +75.438, E3 +19093.976}
ENDSPLINE

SPLINE
SPL {X  -159.644, Y  +366.989, Z    +0.000, E1   +72.058, E3 +19109.503}
ENDSPLINE

SPLINE
SPL {X  -156.933, Y  +346.374, Z    +0.000, E1   +72.645, E3 +19117.393}
SPL {X  -151.144, Y  +325.039, Z    +0.000, E1   +73.323, E3 +19124.072}
SPL {X  -145.016, Y  +309.920, Z    +0.000, E1   +73.647, E3 +19129.866}
SPL {X  -136.944, Y  +294.777, Z    +0.000, E1   +74.219, E3 +19133.168}
SPL {X  -132.590, Y  +287.964, Z    +0.000, E1   +73.910, E3 +19138.912}
SPL {X  -129.541, Y  +283.606, Z    +0.000, E1   +73.551, E3 +19143.553}
SPL {X  -125.403, Y  +278.147, Z    +0.000, E1   +73.063, E3 +19149.360}
SPL {X  -121.908, Y  +273.889, Z    +0.000, E1   +72.578, E3 +19153.906}
SPL {X  -118.941, Y  +270.496, Z    +0.000, E1   +72.188, E3 +19157.394}
SPL {X   -74.907, Y  +236.129, Z    +0.000, E1   +61.720, E3 +19236.008}
ENDSPLINE

SPLINE
SPL {X   -94.059, Y  +248.080, Z    +0.000, E1   +58.275, E3 +19457.701}
SPL {X  -136.558, Y  +294.141, Z    +0.000, E1   +54.887, E3 +19501.555}
SPL {X  -151.843, Y  +327.098, Z    +0.000, E1   +44.118, E3 +19510.915}
SPL {X  -157.484, Y  +349.293, Z    +0.000, E1   +30.654, E3 +19513.954}
SPL {X  -159.556, Y  +365.719, Z    +0.000, E1   +15.845, E3 +19515.147}
SPL {X  -159.982, Y  +375.924, Z    +0.000, E1    +4.476, E3 +19515.448}
SPL {X  -159.990, Y  +379.531, Z    +0.000, E1    -0.039, E3 +19515.475}
SPL {X  -159.990, Y  +382.420, Z    +0.000, E1    -7.600, E3 +19515.504}
SPL {X  -159.990, Y  +387.978, Z    +0.000, E1   -23.882, E3 +19515.672}
SPL {X  -159.990, Y  +396.850, Z    +0.000, E1   -45.459, E3 +19516.259}
SPL {X  -159.990, Y  +409.662, Z    +0.000, E1   -61.705, E3 +19517.688}
SPL {X  -159.990, Y  +426.583, Z    +0.000, E1   -69.729, E3 +19520.802}
SPL {X  -159.990, Y  +451.842, Z    +0.000, E1   -73.935, E3 +19526.729}
SPL {X  -159.990, Y  +521.523, Z    +0.000, E1   -76.035, E3 +19548.989}
SPL {X  -154.459, Y  +718.205, Z    +0.000, E1   -76.329, E3 +19630.784}
SPL {X  -151.356, Y  +728.349, Z    +0.000, E1   -76.056, E3 +19639.000}
SPL {X  -148.399, Y  +736.287, Z    +0.000, E1   -75.788, E3 +19645.878}
SPL {X  -144.005, Y  +746.209, Z    +0.000, E1   -75.396, E3 +19654.994}
SPL {X  -138.117, Y  +757.250, Z    +0.000, E1   -74.803, E3 +19665.884}
SPL {X  -133.491, Y  +764.686, Z    +0.000, E1   -74.276, E3 +19673.625}
SPL {X  -130.530, Y  +769.013, Z    +0.000, E1   -73.929, E3 +19678.207}
SPL {X  -127.734, Y  +772.837, Z    +0.000, E1   -73.601, E3 +19682.259}
SPL {X  -124.765, Y  +776.652, Z    +0.000, E1   -73.233, E3 +19686.294}
SPL {X  -121.376, Y  +780.734, Z    +0.000, E1   -72.804, E3 +19690.555}
SPL {X  -118.281, Y  +784.233, Z    +0.000, E1   -72.371, E3 +19694.124}
SPL {X   -72.391, Y  +819.176, Z    +0.000, E1   -59.867, E3 +19790.009}
ENDSPLINE

SPLINE
SPL {X  -116.241, Y  +786.431, Z    +0.000, E1   -57.120, E3 +20014.452}
SPL {X  -148.710, Y  +735.509, Z    +0.000, E1   -46.282, E3 +20040.184}
SPL {X  -157.559, Y  +704.285, Z    +0.000, E1   -29.037, E3 +20045.514}
SPL {X  -159.709, Y  +685.986, Z    +0.000, E1   -12.810, E3 +20046.845}
SPL {X  -159.990, Y  +674.648, Z    +0.000, E1    -0.349, E3 +20047.105}
SPL {X  -159.990, Y  +672.787, Z    +0.000, E1    +4.022, E3 +20047.117}
SPL {X  -159.990, Y  +669.267, Z    +0.000, E1   +13.665, E3 +20047.188}
SPL {X  -159.990, Y  +663.438, Z    +0.000, E1   +29.379, E3 +20047.458}
SPL {X  -159.990, Y  +655.264, Z    +0.000, E1   +47.291, E3 +20048.075}
SPL {X  -159.990, Y  +645.368, Z    +0.000, E1   +59.257, E3 +20049.318}
SPL {X  -159.990, Y  +624.023, Z    +0.000, E1   +69.513, E3 +20053.443}
SPL {X  -159.990, Y  +543.075, Z    +0.000, E1   +75.590, E3 +20077.091}
SPL {X  -156.121, Y  +342.530, Z    +0.000, E1   +75.868, E3 +20163.737}
SPL {X  -153.498, Y  +332.386, Z    +0.000, E1   +75.628, E3 +20171.742}
ENDSPLINE

SPLINE
SPL {X  -155.252, Y  +338.851, Z    +0.000, E1   +74.632, E3 +20179.120}
SPL {X  -159.103, Y  +360.678, Z    +0.000, E1   +72.233, E3 +20191.445}
ENDSPLINE

SPLINE
SPL {X  -154.371, Y  +335.471, Z    +0.000, E1   +73.016, E3 +20200.016}
SPL {X  -149.938, Y  +321.685, Z    +0.000, E1   +73.398, E3 +20204.710}
SPL {X  -145.016, Y  +309.920, Z    +0.000, E1   +73.647, E3 +20209.231}
SPL {X  -136.944, Y  +294.777, Z    +0.000, E1   +74.219, E3 +20212.533}
SPL {X  -132.590, Y  +287.964, Z    +0.000, E1   +73.910, E3 +20218.277}
SPL {X  -129.541, Y  +283.606, Z    +0.000, E1   +73.551, E3 +20222.918}
SPL {X  -125.403, Y  +278.147, Z    +0.000, E1   +73.063, E3 +20228.725}
SPL {X  -121.908, Y  +273.889, Z    +0.000, E1   +72.578, E3 +20233.271}
SPL {X  -119.156, Y  +270.736, Z    +0.000, E1   +72.213, E3 +20236.521}
SPL {X  -117.531, Y  +268.949, Z    +0.000, E1   +71.964, E3 +20238.337}
SPL {X   -74.907, Y  +236.129, Z    +0.000, E1   +61.720, E3 +20315.373}
ENDSPLINE

SPLINE
SPL {X   -94.059, Y  +248.080, Z    +0.000, E1   +58.275, E3 +20537.066}
SPL {X  -130.769, Y  +285.325, Z    +0.000, E1   +56.495, E3 +20576.943}
SPL {X  -149.689, Y  +321.019, Z    +0.000, E1   +46.817, E3 +20589.027}
SPL {X  -157.484, Y  +349.293, Z    +0.000, E1   +30.654, E3 +20593.319}
SPL {X  -159.556, Y  +365.719, Z    +0.000, E1   +15.845, E3 +20594.512}
SPL {X  -159.982, Y  +375.924, Z    +0.000, E1    +4.476, E3 +20594.813}
SPL {X  -159.990, Y  +379.531, Z    +0.000, E1    -0.039, E3 +20594.840}
SPL {X  -159.990, Y  +382.420, Z    +0.000, E1    -7.600, E3 +20594.869}
SPL {X  -159.990, Y  +386.504, Z    +0.000, E1   -19.860, E3 +20594.974}
SPL {X  -159.990, Y  +392.530, Z    +0.000, E1   -36.133, E3 +20595.289}
SPL {X  -159.990, Y  +400.492, Z    +0.000, E1   -51.837, E3 +20595.942}
SPL {X  -159.990, Y  +409.662, Z    +0.000, E1   -61.705, E3 +20597.053}
SPL {X  -159.990, Y  +434.697, Z    +0.000, E1   -71.504, E3 +20602.073}
SPL {X  -159.990, Y  +521.523, Z    +0.000, E1   -76.035, E3 +20628.354}
SPL {X  -154.459, Y  +718.205, Z    +0.000, E1   -76.329, E3 +20710.149}
SPL {X  -151.356, Y  +728.349, Z    +0.000, E1   -76.056, E3 +20718.365}
SPL {X  -148.399, Y  +736.287, Z    +0.000, E1   -75.788, E3 +20725.243}
SPL {X  -144.005, Y  +746.209, Z    +0.000, E1   -75.396, E3 +20734.359}
SPL {X  -138.117, Y  +757.250, Z    +0.000, E1   -74.803, E3 +20745.249}
SPL {X  -133.491, Y  +764.686, Z    +0.000, E1   -74.276, E3 +20752.990}
SPL {X  -130.530, Y  +769.013, Z    +0.000, E1   -73.929, E3 +20757.572}
SPL {X  -127.734, Y  +772.837, Z    +0.000, E1   -73.601, E3 +20761.624}
SPL {X  -124.765, Y  +776.652, Z    +0.000, E1   -73.233, E3 +20765.659}
SPL {X  -121.376, Y  +780.734, Z    +0.000, E1   -72.804, E3 +20769.920}
SPL {X  -118.281, Y  +784.233, Z    +0.000, E1   -72.371, E3 +20773.489}
SPL {X   -72.391, Y  +819.176, Z    +0.000, E1   -59.867, E3 +20869.374}
ENDSPLINE

SPLINE
SPL {X  -116.241, Y  +786.431, Z    +0.000, E1   -57.120, E3 +21093.817}
SPL {X  -148.710, Y  +735.509, Z    +0.000, E1   -46.282, E3 +21119.549}
SPL {X  -157.559, Y  +704.285, Z    +0.000, E1   -29.037, E3 +21124.879}
SPL {X  -159.709, Y  +685.986, Z    +0.000, E1   -12.810, E3 +21126.210}
SPL {X  -159.990, Y  +674.648, Z    +0.000, E1    -0.349, E3 +21126.470}
SPL {X  -159.990, Y  +672.787, Z    +0.000, E1    +4.022, E3 +21126.482}
SPL {X  -159.990, Y  +669.267, Z    +0.000, E1   +13.665, E3 +21126.553}
SPL {X  -159.990, Y  +663.438, Z    +0.000, E1   +29.379, E3 +21126.823}
SPL {X  -159.990, Y  +655.264, Z    +0.000, E1   +47.291, E3 +21127.440}
SPL {X  -159.990, Y  +645.368, Z    +0.000, E1   +59.257, E3 +21128.684}
SPL {X  -159.990, Y  +624.023, Z    +0.000, E1   +69.513, E3 +21132.808}
SPL {X  -159.990, Y  +543.075, Z    +0.000, E1   +75.590, E3 +21156.456}
SPL {X  -156.121, Y  +342.530, Z    +0.000, E1   +75.868, E3 +21243.103}
SPL {X  -153.498, Y  +332.386, Z    +0.000, E1   +75.628, E3 +21251.107}
ENDSPLINE

SPLINE
SPL {X  -155.252, Y  +338.851, Z    +0.000, E1   +74.632, E3 +21258.485}
SPL {X  -159.103, Y  +360.678, Z    +0.000, E1   +72.233, E3 +21270.810}
ENDSPLINE

SPLINE
SPL {X  -154.371, Y  +335.471, Z    +0.000, E1   +73.016, E3 +21279.381}
SPL {X  -149.938, Y  +321.685, Z    +0.000, E1   +73.398, E3 +21284.075}
SPL {X  -145.016, Y  +309.920, Z    +0.000, E1   +73.647, E3 +21288.596}
SPL {X  -136.944, Y  +294.777, Z    +0.000, E1   +74.219, E3 +21291.898}
SPL {X  -132.590, Y  +287.964, Z    +0.000, E1   +73.910, E3 +21297.642}
SPL {X  -129.541, Y  +283.606, Z    +0.000, E1   +73.551, E3 +21302.283}
SPL {X  -125.403, Y  +278.147, Z    +0.000, E1   +73.063, E3 +21308.090}
SPL {X  -121.908, Y  +273.889, Z    +0.000, E1   +72.578, E3 +21312.636}
SPL {X  -119.156, Y  +270.736, Z    +0.000, E1   +72.213, E3 +21315.886}
SPL {X  -117.531, Y  +268.949, Z    +0.000, E1   +71.964, E3 +21317.702}
SPL {X   -74.907, Y  +236.129, Z    +0.000, E1   +61.720, E3 +21394.738}
ENDSPLINE

SPLINE
SPL {X   -94.059, Y  +248.080, Z    +0.000, E1   +58.275, E3 +21616.431}
SPL {X  -130.769, Y  +285.325, Z    +0.000, E1   +56.495, E3 +21656.308}
SPL {X  -149.689, Y  +321.019, Z    +0.000, E1   +46.817, E3 +21668.392}
SPL {X  -157.484, Y  +349.293, Z    +0.000, E1   +30.654, E3 +21672.684}
SPL {X  -159.556, Y  +365.719, Z    +0.000, E1   +15.845, E3 +21673.877}
SPL {X  -159.982, Y  +375.924, Z    +0.000, E1    +4.476, E3 +21674.178}
SPL {X  -159.990, Y  +379.531, Z    +0.000, E1    -0.039, E3 +21674.205}
SPL {X  -159.990, Y  +382.420, Z    +0.000, E1    -7.600, E3 +21674.234}
SPL {X  -159.990, Y  +386.504, Z    +0.000, E1   -19.860, E3 +21674.339}
SPL {X  -159.990, Y  +392.530, Z    +0.000, E1   -36.133, E3 +21674.654}
SPL {X  -159.990, Y  +400.492, Z    +0.000, E1   -51.837, E3 +21675.307}
SPL {X  -159.990, Y  +409.662, Z    +0.000, E1   -61.705, E3 +21676.418}
SPL {X  -159.990, Y  +434.697, Z    +0.000, E1   -71.504, E3 +21681.438}
SPL {X  -159.990, Y  +521.523, Z    +0.000, E1   -76.035, E3 +21707.719}
SPL {X  -154.459, Y  +718.205, Z    +0.000, E1   -76.329, E3 +21789.514}
SPL {X  -151.356, Y  +728.349, Z    +0.000, E1   -76.056, E3 +21797.730}
SPL {X  -148.399, Y  +736.287, Z    +0.000, E1   -75.788, E3 +21804.608}
SPL {X  -144.005, Y  +746.209, Z    +0.000, E1   -75.396, E3 +21813.724}
SPL {X  -138.117, Y  +757.250, Z    +0.000, E1   -74.803, E3 +21824.614}
SPL {X  -133.491, Y  +764.686, Z    +0.000, E1   -74.276, E3 +21832.355}
SPL {X  -130.530, Y  +769.013, Z    +0.000, E1   -73.929, E3 +21836.937}
SPL {X  -127.734, Y  +772.837, Z    +0.000, E1   -73.601, E3 +21840.989}
SPL {X  -124.765, Y  +776.652, Z    +0.000, E1   -73.233, E3 +21845.024}
SPL {X  -121.376, Y  +780.734, Z    +0.000, E1   -72.804, E3 +21849.285}
SPL {X  -118.281, Y  +784.233, Z    +0.000, E1   -72.371, E3 +21852.854}
SPL {X   -72.391, Y  +819.176, Z    +0.000, E1   -59.867, E3 +21948.740}
ENDSPLINE

SPLINE
SPL {X   -92.809, Y  +806.820, Z    +0.000, E1   -56.994, E3 +22141.535}
SPL {X  -120.521, Y  +781.721, Z    +0.000, E1   -56.766, E3 +22177.633}
SPL {X  -143.482, Y  +747.279, Z    +0.000, E1   -50.227, E3 +22195.646}
SPL {X  -154.118, Y  +719.449, Z    +0.000, E1   -38.836, E3 +22202.226}
SPL {X  -158.958, Y  +694.646, Z    +0.000, E1   -21.132, E3 +22205.077}
SPL {X  -159.960, Y  +679.609, Z    +0.000, E1    -6.021, E3 +22205.777}
SPL {X  -159.990, Y  +674.508, Z    +0.000, E1    -0.018, E3 +22205.836}
SPL {X  -159.990, Y  +672.787, Z    +0.000, E1    +4.022, E3 +22205.847}
SPL {X  -159.990, Y  +669.267, Z    +0.000, E1   +13.665, E3 +22205.918}
SPL {X  -159.990, Y  +665.069, Z    +0.000, E1   +25.376, E3 +22206.090}
SPL {X  -159.990, Y  +657.821, Z    +0.000, E1   +42.408, E3 +22206.592}
SPL {X  -159.990, Y  +645.368, Z    +0.000, E1   +59.257, E3 +22208.049}
SPL {X  -159.990, Y  +624.023, Z    +0.000, E1   +69.513, E3 +22212.173}
SPL {X  -159.990, Y  +543.075, Z    +0.000, E1   +75.590, E3 +22235.821}
SPL {X  -156.121, Y  +342.530, Z    +0.000, E1   +75.868, E3 +22322.468}
SPL {X  -153.865, Y  +333.657, Z    +0.000, E1   +75.438, E3 +22332.072}
ENDSPLINE

SPLINE
SPL {X  -159.103, Y  +360.678, Z    +0.000, E1   +72.233, E3 +22350.175}
ENDSPLINE

SPLINE
SPL {X  -154.371, Y  +335.471, Z    +0.000, E1   +73.016, E3 +22358.746}
SPL {X  -148.318, Y  +317.512, Z    +0.000, E1   +73.488, E3 +22365.067}
SPL {X  -141.230, Y  +302.327, Z    +0.000, E1   +73.933, E3 +22369.621}
SPL {X  -135.697, Y  +292.747, Z    +0.000, E1   +74.259, E3 +22371.979}
SPL {X  -132.590, Y  +287.964, Z    +0.000, E1   +73.910, E3 +22377.007}
SPL {X  -129.541, Y  +283.606, Z    +0.000, E1   +73.551, E3 +22381.648}
SPL {X  -126.457, Y  +279.493, Z    +0.000, E1   +73.175, E3 +22386.047}
SPL {X  -122.770, Y  +274.912, Z    +0.000, E1   +72.712, E3 +22390.902}
SPL {X  -119.156, Y  +270.736, Z    +0.000, E1   +72.213, E3 +22395.251}
SPL {X  -117.531, Y  +268.949, Z    +0.000, E1   +71.964, E3 +22397.067}
SPL {X   -74.907, Y  +236.129, Z    +0.000, E1   +61.720, E3 +22474.103}
SPL {X   -72.759, Y  +235.012, Z    +0.000, E1   +56.036, E3 +22645.780}
ENDSPLINE

SPLINE
SPL {X  -110.316, Y  +261.624, Z    +0.000, E1   +58.739, E3 +22717.853}
SPL {X  -136.558, Y  +294.141, Z    +0.000, E1   +54.887, E3 +22739.650}
SPL {X  -153.807, Y  +333.452, Z    +0.000, E1   +40.945, E3 +22750.047}
SPL {X  -158.168, Y  +353.421, Z    +0.000, E1   +27.296, E3 +22752.441}
SPL {X  -159.556, Y  +365.719, Z    +0.000, E1   +15.845, E3 +22753.242}
SPL {X  -159.982, Y  +375.924, Z    +0.000, E1    +4.476, E3 +22753.543}
SPL {X  -159.990, Y  +379.800, Z    +0.000, E1    -0.377, E3 +22753.572}
SPL {X  -159.990, Y  +383.422, Z    +0.000, E1   -10.730, E3 +22753.615}
SPL {X  -159.990, Y  +387.978, Z    +0.000, E1   -23.882, E3 +22753.767}
SPL {X  -159.990, Y  +394.494, Z    +0.000, E1   -40.961, E3 +22754.148}
SPL {X  -159.990, Y  +400.492, Z    +0.000, E1   -51.837, E3 +22754.672}
SPL {X  -159.990, Y  +409.662, Z    +0.000, E1   -61.705, E3 +22755.783}
SPL {X  -159.990, Y  +434.697, Z    +0.000, E1   -71.504, E3 +22760.803}
SPL {X  -159.990, Y  +521.523, Z    +0.000, E1   -76.035, E3 +22787.084}
SPL {X  -154.459, Y  +718.205, Z    +0.000, E1   -76.329, E3 +22868.879}
SPL {X  -151.356, Y  +728.349, Z    +0.000, E1   -76.056, E3 +22877.095}
SPL {X  -147.124, Y  +739.360, Z    +0.000, E1   -75.690, E3 +22886.691}
SPL {X  -142.861, Y  +748.524, Z    +0.000, E1   -75.261, E3 +22895.376}
SPL {X  -138.117, Y  +757.250, Z    +0.000, E1   -74.803, E3 +22903.980}
SPL {X  -133.491, Y  +764.686, Z    +0.000, E1   -74.276, E3 +22911.720}
SPL {X  -130.530, Y  +769.013, Z    +0.000, E1   -73.929, E3 +22916.302}
SPL {X  -127.734, Y  +772.837, Z    +0.000, E1   -73.601, E3 +22920.355}
SPL {X  -124.765, Y  +776.652, Z    +0.000, E1   -73.233, E3 +22924.389}
SPL {X  -121.376, Y  +780.734, Z    +0.000, E1   -72.804, E3 +22928.650}
SPL {X  -118.281, Y  +784.233, Z    +0.000, E1   -72.371, E3 +22932.219}
SPL {X   -72.391, Y  +819.176, Z    +0.000, E1   -59.867, E3 +23028.105}
ENDSPLINE

SPLINE
SPL {X  -116.241, Y  +786.431, Z    +0.000, E1   -57.120, E3 +23252.547}
SPL {X  -148.710, Y  +735.509, Z    +0.000, E1   -46.282, E3 +23278.280}
SPL {X  -157.559, Y  +704.285, Z    +0.000, E1   -29.037, E3 +23283.609}
SPL {X  -159.430, Y  +689.871, Z    +0.000, E1   -16.582, E3 +23284.759}
SPL {X  -159.960, Y  +679.609, Z    +0.000, E1    -6.021, E3 +23285.142}
SPL {X  -159.990, Y  +674.508, Z    +0.000, E1    -0.018, E3 +23285.201}
SPL {X  -159.990, Y  +672.787, Z    +0.000, E1    +4.022, E3 +23285.213}
SPL {X  -159.990, Y  +669.267, Z    +0.000, E1   +13.665, E3 +23285.283}
SPL {X  -159.990, Y  +665.069, Z    +0.000, E1   +25.376, E3 +23285.455}
SPL {X  -159.990, Y  +657.821, Z    +0.000, E1   +42.408, E3 +23285.957}
SPL {X  -159.990, Y  +645.368, Z    +0.000, E1   +59.257, E3 +23287.414}
SPL {X  -159.990, Y  +624.023, Z    +0.000, E1   +69.513, E3 +23291.539}
SPL {X  -159.990, Y  +543.075, Z    +0.000, E1   +75.590, E3 +23315.186}
SPL {X  -156.121, Y  +342.530, Z    +0.000, E1   +75.868, E3 +23401.833}
SPL {X  -153.865, Y  +333.657, Z    +0.000, E1   +75.438, E3 +23411.437}
ENDSPLINE

SPLINE
SPL {X  -159.644, Y  +366.989, Z    +0.000, E1   +72.058, E3 +23426.964}
ENDSPLINE

SPLINE
SPL {X  -156.933, Y  +346.374, Z    +0.000, E1   +72.645, E3 +23434.853}
SPL {X  -151.144, Y  +325.039, Z    +0.000, E1   +73.323, E3 +23441.533}
SPL {X  -145.016, Y  +309.920, Z    +0.000, E1   +73.647, E3 +23447.326}
SPL {X  -136.944, Y  +294.777, Z    +0.000, E1   +74.219, E3 +23450.628}
SPL {X  -132.590, Y  +287.964, Z    +0.000, E1   +73.910, E3 +23456.372}
SPL {X  -129.541, Y  +283.606, Z    +0.000, E1   +73.551, E3 +23461.013}
SPL {X  -125.403, Y  +278.147, Z    +0.000, E1   +73.063, E3 +23466.820}
SPL {X  -121.908, Y  +273.889, Z    +0.000, E1   +72.578, E3 +23471.366}
SPL {X  -118.941, Y  +270.496, Z    +0.000, E1   +72.188, E3 +23474.855}
SPL {X   -74.907, Y  +236.129, Z    +0.000, E1   +61.720, E3 +23553.468}
ENDSPLINE

SPLINE
SPL {X   -94.059, Y  +248.080, Z    +0.000, E1   +58.275, E3 +23775.161}
SPL {X  -136.558, Y  +294.141, Z    +0.000, E1   +54.887, E3 +23819.015}
SPL {X  -151.843, Y  +327.098, Z    +0.000, E1   +44.118, E3 +23828.375}
SPL {X  -157.484, Y  +349.293, Z    +0.000, E1   +30.654, E3 +23831.414}
SPL {X  -159.556, Y  +365.719, Z    +0.000, E1   +15.845, E3 +23832.607}
SPL {X  -159.982, Y  +375.924, Z    +0.000, E1    +4.476, E3 +23832.909}
SPL {X  -159.990, Y  +379.531, Z    +0.000, E1    -0.039, E3 +23832.936}
SPL {X  -159.990, Y  +382.420, Z    +0.000, E1    -7.600, E3 +23832.964}
SPL {X  -159.990, Y  +386.504, Z    +0.000, E1   -19.860, E3 +23833.069}
SPL {X  -159.990, Y  +392.530, Z    +0.000, E1   -36.133, E3 +23833.385}
SPL {X  -159.990, Y  +400.492, Z    +0.000, E1   -51.837, E3 +23834.037}
SPL {X  -159.990, Y  +409.662, Z    +0.000, E1   -61.705, E3 +23835.149}
SPL {X  -159.990, Y  +434.697, Z    +0.000, E1   -71.504, E3 +23840.168}
SPL {X  -159.990, Y  +521.523, Z    +0.000, E1   -76.035, E3 +23866.449}
SPL {X  -154.459, Y  +718.205, Z    +0.000, E1   -76.329, E3 +23948.244}
SPL {X  -151.356, Y  +728.349, Z    +0.000, E1   -76.056, E3 +23956.460}
SPL {X  -148.399, Y  +736.287, Z    +0.000, E1   -75.788, E3 +23963.339}
SPL {X  -144.005, Y  +746.209, Z    +0.000, E1   -75.396, E3 +23972.455}
SPL {X  -138.117, Y  +757.250, Z    +0.000, E1   -74.803, E3 +23983.345}
SPL {X  -133.491, Y  +764.686, Z    +0.000, E1   -74.276, E3 +23991.086}
SPL {X  -128.839, Y  +771.354, Z    +0.000, E1   -73.759, E3 +23998.104}
SPL {X  -123.568, Y  +778.125, Z    +0.000, E1   -73.105, E3 +24005.276}
SPL {X  -118.985, Y  +783.455, Z    +0.000, E1   -72.490, E3 +24010.783}
SPL {X   -72.391, Y  +819.176, Z    +0.000, E1   -59.867, E3 +24107.470}
ENDSPLINE

SPLINE
SPL {X   -92.809, Y  +806.820, Z    +0.000, E1   -56.994, E3 +24300.265}
SPL {X  -120.521, Y  +781.721, Z    +0.000, E1   -56.766, E3 +24336.364}
SPL {X  -143.482, Y  +747.279, Z    +0.000, E1   -50.227, E3 +24354.377}
SPL {X  -154.118, Y  +719.449, Z    +0.000, E1   -38.836, E3 +24360.956}
SPL {X  -158.281, Y  +699.823, Z    +0.000, E1   -25.469, E3 +24363.420}
SPL {X  -159.709, Y  +685.986, Z    +0.000, E1   -12.810, E3 +24364.306}
SPL {X  -159.990, Y  +674.648, Z    +0.000, E1    -0.349, E3 +24364.565}
SPL {X  -159.990, Y  +672.787, Z    +0.000, E1    +4.022, E3 +24364.578}
SPL {X  -159.990, Y  +669.267, Z    +0.000, E1   +13.665, E3 +24364.648}
SPL {X  -159.990, Y  +665.069, Z    +0.000, E1   +25.376, E3 +24364.820}
SPL {X  -159.990, Y  +657.821, Z    +0.000, E1   +42.408, E3 +24365.322}
SPL {X  -159.990, Y  +645.368, Z    +0.000, E1   +59.257, E3 +24366.779}
SPL {X  -159.990, Y  +624.023, Z    +0.000, E1   +69.513, E3 +24370.904}
SPL {X  -159.990, Y  +543.075, Z    +0.000, E1   +75.590, E3 +24394.552}
SPL {X  -156.121, Y  +342.530, Z    +0.000, E1   +75.868, E3 +24481.198}
SPL {X  -153.865, Y  +333.657, Z    +0.000, E1   +75.438, E3 +24490.802}
ENDSPLINE

SPLINE
SPL {X  -159.644, Y  +366.989, Z    +0.000, E1   +72.058, E3 +24506.329}
ENDSPLINE

SPLINE
SPL {X  -156.933, Y  +346.374, Z    +0.000, E1   +72.645, E3 +24514.218}
SPL {X  -151.144, Y  +325.039, Z    +0.000, E1   +73.323, E3 +24520.898}
SPL {X  -145.016, Y  +309.920, Z    +0.000, E1   +73.647, E3 +24526.691}
SPL {X  -136.944, Y  +294.777, Z    +0.000, E1   +74.219, E3 +24529.993}
SPL {X  -132.590, Y  +287.964, Z    +0.000, E1   +73.910, E3 +24535.737}
SPL {X  -129.541, Y  +283.606, Z    +0.000, E1   +73.551, E3 +24540.378}
SPL {X  -126.457, Y  +279.493, Z    +0.000, E1   +73.175, E3 +24544.777}
SPL {X  -122.770, Y  +274.912, Z    +0.000, E1   +72.712, E3 +24549.632}
SPL {X  -119.156, Y  +270.736, Z    +0.000, E1   +72.213, E3 +24553.982}
SPL {X  -117.531, Y  +268.949, Z    +0.000, E1   +71.964, E3 +24555.797}
SPL {X   -74.907, Y  +236.129, Z    +0.000, E1   +61.720, E3 +24632.833}
ENDSPLINE

SPLINE
SPL {X   -94.059, Y  +248.080, Z    +0.000, E1   +58.275, E3 +24854.526}
SPL {X  -130.769, Y  +285.325, Z    +0.000, E1   +56.495, E3 +24894.403}
SPL {X  -149.689, Y  +321.019, Z    +0.000, E1   +46.817, E3 +24906.487}
SPL {X  -157.484, Y  +349.293, Z    +0.000, E1   +30.654, E3 +24910.779}
SPL {X  -159.556, Y  +365.719, Z    +0.000, E1   +15.845, E3 +24911.972}
SPL {X  -159.982, Y  +375.924, Z    +0.000, E1    +4.476, E3 +24912.274}
SPL {X  -159.990, Y  +379.531, Z    +0.000, E1    -0.039, E3 +24912.301}
SPL {X  -159.990, Y  +382.420, Z    +0.000, E1    -7.600, E3 +24912.329}
SPL {X  -159.990, Y  +386.504, Z    +0.000, E1   -19.860, E3 +24912.434}
SPL {X  -159.990, Y  +392.530, Z    +0.000, E1   -36.133, E3 +24912.750}
SPL {X  -159.990, Y  +400.492, Z    +0.000, E1   -51.837, E3 +24913.402}
SPL {X  -159.990, Y  +409.662, Z    +0.000, E1   -61.705, E3 +24914.514}
SPL {X  -159.990, Y  +434.697, Z    +0.000, E1   -71.504, E3 +24919.534}
SPL {X  -159.990, Y  +521.523, Z    +0.000, E1   -76.035, E3 +24945.814}
SPL {X  -154.459, Y  +718.205, Z    +0.000, E1   -76.329, E3 +25027.609}
SPL {X  -151.356, Y  +728.349, Z    +0.000, E1   -76.056, E3 +25035.825}
SPL {X  -148.399, Y  +736.287, Z    +0.000, E1   -75.788, E3 +25042.704}
SPL {X  -144.005, Y  +746.209, Z    +0.000, E1   -75.396, E3 +25051.820}
SPL {X  -138.117, Y  +757.250, Z    +0.000, E1   -74.803, E3 +25062.710}
SPL {X  -133.491, Y  +764.686, Z    +0.000, E1   -74.276, E3 +25070.451}
SPL {X  -130.530, Y  +769.013, Z    +0.000, E1   -73.929, E3 +25075.032}
SPL {X  -127.734, Y  +772.837, Z    +0.000, E1   -73.601, E3 +25079.085}
SPL {X  -124.765, Y  +776.652, Z    +0.000, E1   -73.233, E3 +25083.119}
SPL {X  -121.376, Y  +780.734, Z    +0.000, E1   -72.804, E3 +25087.381}
SPL {X  -118.281, Y  +784.233, Z    +0.000, E1   -72.371, E3 +25090.949}
SPL {X   -72.391, Y  +819.176, Z    +0.000, E1   -59.867, E3 +25186.835}
ENDSPLINE

SPLINE
SPL {X  -116.241, Y  +786.431, Z    +0.000, E1   -57.120, E3 +25411.277}
SPL {X  -148.710, Y  +735.509, Z    +0.000, E1   -46.282, E3 +25437.010}
SPL {X  -157.559, Y  +704.285, Z    +0.000, E1   -29.037, E3 +25442.339}
SPL {X  -159.709, Y  +685.986, Z    +0.000, E1   -12.810, E3 +25443.671}
SPL {X  -159.990, Y  +674.648, Z    +0.000, E1    -0.349, E3 +25443.930}
SPL {X  -159.990, Y  +672.787, Z    +0.000, E1    +4.022, E3 +25443.943}
SPL {X  -159.990, Y  +669.267, Z    +0.000, E1   +13.665, E3 +25444.013}
SPL {X  -159.990, Y  +663.438, Z    +0.000, E1   +29.379, E3 +25444.284}
SPL {X  -159.990, Y  +655.264, Z    +0.000, E1   +47.291, E3 +25444.900}
SPL {X  -159.990, Y  +645.368, Z    +0.000, E1   +59.257, E3 +25446.144}
SPL {X  -159.990, Y  +624.023, Z    +0.000, E1   +69.513, E3 +25450.269}
SPL {X  -159.990, Y  +543.075, Z    +0.000, E1   +75.590, E3 +25473.917}
SPL {X  -156.121, Y  +342.530, Z    +0.000, E1   +75.868, E3 +25560.563}
SPL {X  -153.498, Y  +332.386, Z    +0.000, E1   +75.628, E3 +25568.567}
ENDSPLINE

SPLINE
SPL {X  -155.252, Y  +338.851, Z    +0.000, E1   +74.632, E3 +25575.946}
SPL {X  -159.103, Y  +360.678, Z    +0.000, E1   +72.233, E3 +25588.271}
ENDSPLINE

SPLINE
SPL {X  -154.371, Y  +335.471, Z    +0.000, E1   +73.016, E3 +25596.841}
SPL {X  -149.938, Y  +321.685, Z    +0.000, E1   +73.398, E3 +25601.536}
SPL {X  -145.016, Y  +309.920, Z    +0.000, E1   +73.647, E3 +25606.057}
SPL {X  -136.944, Y  +294.777, Z    +0.000, E1   +74.219, E3 +25609.358}
SPL {X  -132.590, Y  +287.964, Z    +0.000, E1   +73.910, E3 +25615.103}
SPL {X  -129.541, Y  +283.606, Z    +0.000, E1   +73.551, E3 +25619.743}
SPL {X  -125.403, Y  +278.147, Z    +0.000, E1   +73.063, E3 +25625.550}
SPL {X  -121.908, Y  +273.889, Z    +0.000, E1   +72.578, E3 +25630.097}
SPL {X  -119.156, Y  +270.736, Z    +0.000, E1   +72.213, E3 +25633.347}
SPL {X  -117.531, Y  +268.949, Z    +0.000, E1   +71.964, E3 +25635.162}
SPL {X   -74.907, Y  +236.129, Z    +0.000, E1   +61.720, E3 +25712.198}
ENDSPLINE

SPLINE
SPL {X   -94.059, Y  +248.080, Z    +0.000, E1   +58.275, E3 +25933.891}
SPL {X  -130.769, Y  +285.325, Z    +0.000, E1   +56.495, E3 +25973.768}
SPL {X  -149.689, Y  +321.019, Z    +0.000, E1   +46.817, E3 +25985.852}
SPL {X  -157.484, Y  +349.293, Z    +0.000, E1   +30.654, E3 +25990.145}
SPL {X  -159.556, Y  +365.719, Z    +0.000, E1   +15.845, E3 +25991.337}
SPL {X  -159.982, Y  +375.924, Z    +0.000, E1    +4.476, E3 +25991.639}
SPL {X  -159.990, Y  +379.531, Z    +0.000, E1    -0.039, E3 +25991.666}
SPL {X  -159.990, Y  +382.420, Z    +0.000, E1    -7.600, E3 +25991.694}
SPL {X  -159.990, Y  +386.504, Z    +0.000, E1   -19.860, E3 +25991.800}
SPL {X  -159.990, Y  +392.530, Z    +0.000, E1   -36.133, E3 +25992.115}
SPL {X  -159.990, Y  +400.492, Z    +0.000, E1   -51.837, E3 +25992.768}
SPL {X  -159.990, Y  +409.662, Z    +0.000, E1   -61.705, E3 +25993.879}
SPL {X  -159.990, Y  +434.697, Z    +0.000, E1   -71.504, E3 +25998.899}
SPL {X  -159.990, Y  +521.523, Z    +0.000, E1   -76.035, E3 +26025.179}
SPL {X  -154.459, Y  +718.205, Z    +0.000, E1   -76.329, E3 +26106.975}
SPL {X  -151.356, Y  +728.349, Z    +0.000, E1   -76.056, E3 +26115.190}
SPL {X  -148.399, Y  +736.287, Z    +0.000, E1   -75.788, E3 +26122.069}
SPL {X  -144.005, Y  +746.209, Z    +0.000, E1   -75.396, E3 +26131.185}
SPL {X  -138.117, Y  +757.250, Z    +0.000, E1   -74.803, E3 +26142.075}
SPL {X  -133.491, Y  +764.686, Z    +0.000, E1   -74.276, E3 +26149.816}
SPL {X  -128.839, Y  +771.354, Z    +0.000, E1   -73.759, E3 +26156.834}
SPL {X  -123.568, Y  +778.125, Z    +0.000, E1   -73.105, E3 +26164.006}
SPL {X  -118.985, Y  +783.455, Z    +0.000, E1   -72.490, E3 +26169.514}
SPL {X   -72.391, Y  +819.176, Z    +0.000, E1   -59.867, E3 +26266.200}
ENDSPLINE

SPLINE
SPL {X   -92.809, Y  +806.820, Z    +0.000, E1   -56.994, E3 +26458.995}
SPL {X  -120.521, Y  +781.721, Z    +0.000, E1   -56.766, E3 +26495.094}
SPL {X  -143.482, Y  +747.279, Z    +0.000, E1   -50.227, E3 +26513.107}
SPL {X  -154.118, Y  +719.449, Z    +0.000, E1   -38.836, E3 +26519.686}
SPL {X  -158.958, Y  +694.646, Z    +0.000, E1   -21.132, E3 +26522.537}
SPL {X  -159.960, Y  +679.609, Z    +0.000, E1    -6.021, E3 +26523.237}
SPL {X  -159.990, Y  +674.508, Z    +0.000, E1    -0.018, E3 +26523.296}
SPL {X  -159.990, Y  +672.787, Z    +0.000, E1    +4.022, E3 +26523.308}
SPL {X  -159.990, Y  +669.267, Z    +0.000, E1   +13.665, E3 +26523.378}
SPL {X  -159.990, Y  +663.438, Z    +0.000, E1   +29.379, E3 +26523.649}
SPL {X  -159.990, Y  +655.264, Z    +0.000, E1   +47.291, E3 +26524.266}
SPL {X  -159.990, Y  +645.368, Z    +0.000, E1   +59.257, E3 +26525.509}
SPL {X  -159.990, Y  +624.023, Z    +0.000, E1   +69.513, E3 +26529.634}
SPL {X  -159.990, Y  +543.075, Z    +0.000, E1   +75.590, E3 +26553.282}
SPL {X  -156.121, Y  +342.530, Z    +0.000, E1   +75.868, E3 +26639.928}
SPL {X  -153.498, Y  +332.386, Z    +0.000, E1   +75.628, E3 +26647.932}
ENDSPLINE

SPLINE
SPL {X  -155.252, Y  +338.851, Z    +0.000, E1   +74.632, E3 +26655.311}
SPL {X  -159.103, Y  +360.678, Z    +0.000, E1   +72.233, E3 +26667.636}
ENDSPLINE

